ESR_mon_R4 monitores up to 4 Real inputs and reports changes with time stamd and adress label.
the module checks 4 inputs for a change of more than the specified sensitivity S and reports all changes with time and adress stamp to the output.

*)
(* read system timer *)
tx := DWORD_TO_TIME(T_PLC_MS());
P0 := ADR(R0);
P1 := ADR(R1);
P2 := ADR(R2);
P3 := ADR(R3);

ESR_Flag := FALSE;
esr_out[3].typ := 0;
esr_out[2].typ := 0;
esr_out[1].typ := 0;
esr_out[0].typ := 0;
cnt := 0;

(* check if inputs have chaged and fill buffer *)
IF DIFFER(R0,  X0, S0) THEN
	esr_out[cnt].typ := 20;
	esr_out[cnt].adress := a0;
	esr_out[cnt].DS := DT_in;
	esr_out[cnt].TS := TX;
	esr_out[cnt].data[0] := Byte_of_Dword(P0^,0);
	esr_out[cnt].data[1] := Byte_of_Dword(P0^,1);
	esr_out[cnt].data[2] := Byte_of_Dword(P0^,2);
	esr_out[cnt].data[3] := Byte_of_Dword(P0^,3);
	X0 := R0;
	cnt := cnt + 1;
	esr_flag := TRUE;
END_IF;
IF differ(R1,  X1, S1) THEN
	esr_out[cnt].typ := 20;
	esr_out[cnt].adress := a1;
	esr_out[cnt].DS := DT_in;
	esr_out[cnt].TS := TX;
	esr_out[cnt].data[0] := Byte_of_Dword(P1^,0);
	esr_out[cnt].data[1] := Byte_of_Dword(P1^,1);
	esr_out[cnt].data[2] := Byte_of_Dword(P1^,2);
	esr_out[cnt].data[3] := Byte_of_Dword(P1^,3);
	X1 := R1;
	cnt := cnt + 1;
	esr_flag := TRUE;
END_IF;
IF differ(R2,  X2, S2) THEN
	esr_out[cnt].typ := 20;
	esr_out[cnt].adress := a2;
	esr_out[cnt].DS := DT_in;
	esr_out[cnt].TS := TX;
	esr_out[cnt].data[0] := Byte_of_Dword(P2^,0);
	esr_out[cnt].data[1] := Byte_of_Dword(P2^,1);
	esr_out[cnt].data[2] := Byte_of_Dword(P2^,2);
	esr_out[cnt].data[3] := Byte_of_Dword(P2^,3);
	X2 := R2;
	cnt := cnt + 1;
	esr_flag := TRUE;
END_IF;
IF DIFFER(R3,  X3, S3) THEN
	esr_out[cnt].typ := 20;
	esr_out[cnt].adress := a3;
	esr_out[cnt].DS := DT_in;
	esr_out[cnt].TS := TX;
	esr_out[cnt].data[0] := Byte_of_Dword(P3^,0);
	esr_out[cnt].data[1] := Byte_of_Dword(P3^,1);
	esr_out[cnt].data[2] := Byte_of_Dword(P3^,2);
	esr_out[cnt].data[3] := Byte_of_Dword(P3^,3);
	X3 := R3;
	cnt := cnt + 1;
	esr_flag := TRUE;
END_IF;


(* revision history
hm	26. jan 2007	rev 1.0
	original version

hm	17. sep. 2007		rev 1.1
	replaced time() with T_PLC_MS() for compatibility reasons

hm	8. dec. 2007		rev 1.2
	corrected an error while esr typ would not be set

hm	16. mar. 2008		rev 1.3
	deleted wrong conversion real_to_dword

*)
END_FUNCTION_BLOCK

(* POU ESR_MON_X8, ST *)
FUNCTION_BLOCK ESR_MON_X8
VAR_INPUT
	s0, s1, s2, s3, s4, s5, s6, s7 : BYTE;
	DT_in : DT;
	Mode : BYTE := 3;
END_VAR
VAR_INPUT CONSTANT
	a0, a1, a2, a3, a4, a5, a6, a7 : STRING(10);
END_VAR
VAR_OUTPUT
	ESR_Out: ARRAY [0..3] OF esr_data;
	ESR_Flag : BOOL;
END_VAR
VAR
	x0, x1, x2, x3, x4, x5, x6, x7 : BYTE;
	tx: TIME;
	cnt : INT;
END_VAR

(*
version 1.1	17 sep 2007
programmer 	hugo
tested by		tobias

ESR_MON_X8 is a status and error collector.
the module checks 8 status inputs for a change and reports up to 4 input changes with time and adress stamp to the output.
the mode can be 
1 for error only
2 for error and status
3 for error, status and debug
the adress label of the 8 inputs can be configured individually.
*)
(* read system timer *)
tx := DWORD_TO_TIME(T_PLC_MS());

ESR_Flag := FALSE;
esr_out[3].typ := 0;
esr_out[2].typ := 0;
esr_out[1].typ := 0;
esr_out[0].typ := 0;
cnt := 0;


(* check if inputs have chaged and fill buffer *)
IF s0 <> X0 AND ((s0 < 100) OR (S0 > 99 AND S0 < 200 AND mode >= 2) OR (S0 > 199 AND mode = 3)) THEN
	esr_out[cnt] := status_to_ESR(s0, a0, DT_in, TX);
	X0 := S0;
	cnt := cnt + 1;
	esr_flag := TRUE;
END_IF;
IF s1 <> X1 AND ((s1 < 100) OR (S1 > 99 AND S1 < 200 AND mode >= 2) OR (S1 > 199 AND mode = 3)) THEN
	esr_out[cnt] := status_to_ESR(s1, a1, DT_in, TX);
	X1 := S1;
	cnt := cnt + 1;
	esr_flag := TRUE;
END_IF;
IF s2 <> X2 AND ((s2 < 100) OR (S2 > 99 AND S2 < 200 AND mode >= 2) OR (S2 > 199 AND mode = 3)) THEN
	esr_out[cnt] := status_to_ESR(s2, a2, DT_in, TX);
	X2 := S2;
	cnt := cnt + 1;
	esr_flag := TRUE;
END_IF;
IF s3 <> X3 AND ((s3 < 100) OR (S3 > 99 AND S3 < 200 AND mode >= 2) OR (S3 > 199 AND mode = 3)) THEN
	esr_out[cnt] := status_to_ESR(s3, a3, DT_in, TX);
	X3 := S3;
	cnt := cnt + 1;
	esr_flag := TRUE;
END_IF;
IF cnt < 4 AND s4 <> X4 AND ((s4 < 100) OR (S4 > 99 AND S4 < 200 AND mode >= 2) OR (S4 > 199 AND mode = 3)) THEN
	esr_out[cnt] := status_to_ESR(s4, a4, DT_in, TX);
	X4 := S4;
	cnt := cnt + 1;
	esr_flag := TRUE;
END_IF;
IF cnt < 4 AND s5 <> X5 AND ((s5 < 100) OR (S5 > 99 AND S5 < 200 AND mode >= 2) OR (S5 > 199 AND mode = 3)) THEN
	esr_out[cnt] := status_to_ESR(s5, a5, DT_in, TX);
	X5 := S5;
	cnt := cnt + 1;
	esr_flag := TRUE;
END_IF;
IF cnt < 4 AND s6 <> X6 AND ((s6 < 100) OR (S6 > 99 AND S6 < 200 AND mode >= 2) OR (S6 > 199 AND mode = 3)) THEN
	esr_out[cnt] := status_to_ESR(s6, a6, DT_in, TX);
	X6 := S6;
	cnt := cnt + 1;
	esr_flag := TRUE;
END_IF;
IF cnt < 4 AND s7 <> X7 AND ((s7 < 100) OR (S7 > 99 AND S7 < 200 AND mode >= 2) OR (S7 > 199 AND mode = 3)) THEN
	esr_out[cnt] := status_to_ESR(s7, a7, DT_in, TX);
	X7 := S7;
	cnt := cnt + 1;
	esr_flag := TRUE;
END_IF;


(* revision history
hm	26. jan 2007		rev 1.0
	original version

hm	17. sep 2007	rev 1.1
	replaced time() with T_PLC_MS() for compatibility reasons
	
*)
END_FUNCTION_BLOCK

(* POU STATUS_TO_ESR, ST *)
FUNCTION STATUS_TO_ESR : esr_data
VAR_INPUT
	status : BYTE;
	adress : STRING(10);
	DT_in : DT;
	TS : TIME;
END_VAR
VAR
END_VAR

(*
version 1.0	6 oct 2006
programmer 	hugo
tested by		tobias

status_to_esr creates esr data from a status byte.

*)
IF status < 100 THEN
	status_to_ESR.typ := 1;
ELSIF status < 200 THEN
	status_to_ESR.typ := 2;
ELSE
	status_to_ESR.typ := 3;
END_IF;
status_to_ESR.adress:= adress;
status_to_ESR.DS := DT_in;
status_to_ESR.TS := TS;
status_to_ESR.data[0] := status;
END_FUNCTION

(* POU EXEC, ST *)
FUNCTION EXEC : STRING(STRING_LENGTH)
VAR_INPUT
	str : STRING(STRING_LENGTH);
END_VAR
VAR
	pos: INT;
	R1: REAL;
	R2: REAL;
	operator: STRING(10);
END_VAR

(*
version 1.4	29. mar. 2008
programmer 	hugo
tested by		tobias

exec executes a mathematical term and returns the result as a string
the term can only be a simple term without brackets and only one operator
allowed operastors are: (+, -, *, /, ^, sqrt, sin, cos, tan).

*)
(* extract both numbers and operator *)
EXEC := UPPERCASE(TRIM(str));

pos := FINDB_NONUM(EXEC);
IF pos > 1 THEN R1 := STRING_TO_REAL(LEFT(EXEC,pos-1)); END_IF;
R2 := STRING_TO_REAL(RIGHT(EXEC,LEN(EXEC)-pos));
EXEC := LEFT(EXEC,pos);
pos := FINDB_NUM(EXEC);
operator := RIGHT(EXEC,LEN(EXEC) - pos);
IF operator = '' AND LEN(str) = 0 THEN
	EXEC := '';
	RETURN;
ELSIF operator = '' THEN
	EXEC := str;
	RETURN;
END_IF;
IF operator = '^' THEN
	EXEC := REAL_TO_STRING(EXPT(R1, R2));
ELSIF operator = 'SQRT' THEN
	EXEC := REAL_TO_STRING(SQRT(R2));
ELSIF operator = 'SIN' THEN
	EXEC := REAL_TO_STRING(SIN(r2));
ELSIF operator = 'COS' THEN
	EXEC := REAL_TO_STRING(COS(r2));
ELSIF operator = 'TAN' THEN
	EXEC := REAL_TO_STRING(TAN(R2));
ELSIF operator = '*' THEN
	EXEC := REAL_TO_STRING(R1 * R2);
ELSIF operator = '/' THEN
	IF R2 <> 0 THEN EXEC := REAL_TO_STRING(R1 / R2); ELSE EXEC := 'ERROR'; END_IF;
ELSIF operator = '+' THEN
	EXEC := REAL_TO_STRING(r1 + r2);
ELSIF operator = '-' THEN
	EXEC := REAL_TO_STRING(r1 - r2);
ELSE
	EXEC := 'ERROR';
END_IF;

IF EXEC = 'ERROR' THEN
	RETURN;
(* some systems deliver integer instead of real *)
ELSIF FIND(EXEC,'.') = 0 THEN
	EXEC := CONCAT(EXEC, '.0');
(* some systems deliver n. instead of n.0 ! *)
ELSIF RIGHT(EXEC,1) = '.' THEN
	EXEC := CONCAT(EXEC,'0');
END_IF;


(* revision history

hm 	6.feb 2007		rev 1.1
	cos has to be written in uppercase
	divide by 0 will return an error

hm	5. mar. 2008	rev 1.2
	add a 0 to the string if a '.' is at the end of the string

hm	20. mar. 2008	rev 1.3
	make sure the function always returns a real value in the form of x.y

hm	29. mar. 2008	rev 1.4
	changed STRING to STRING(STRING_LENGTH)
*)
END_FUNCTION

(* POU UPPERCASE, ST *)
FUNCTION UPPERCASE : STRING(STRING_LENGTH)
VAR_INPUT
	str : STRING(STRING_LENGTH);
END_VAR
VAR
	pt : POINTER TO BYTE;
	pos: INT;
	l: INT;
END_VAR

(*
version 1.3	29. mar. 2008
programmer 	hugo
tested by	tobias

uppercase returns str while all letters a..z and ä,ö,ü are converted to uppercase

*)
pt := ADR(UPPERCASE);
UPPERCASE := str;
l := LEN(str);
FOR pos := 1 TO l DO
	pt^ := TO_UPPER(pt^);
	pt := pt + 1;
END_FOR;

(* revision histroy
hm	6. oct. 2006	rev 1.0
	original release

hm	4. feb. 2008	rev 1.1
	improved performance
	added Ä,Ö,Ü

hm	6. mar. 2008	rev 1.2
	added support for exteded Ascii

hm	29. mar. 2008	rev 1.3
	changed STRING to STRING(STRING_LENGTH)

*)	
END_FUNCTION

(* POU TRIM, ST *)
FUNCTION TRIM : STRING(STRING_LENGTH)
VAR_INPUT
	str : STRING(STRING_LENGTH);
END_VAR
VAR
	pos: INT;
END_VAR

(*
version 1.2	29. mar. 2008
programmer 	hugo
tested by	tobias

the function deletes all blanks within a string.

*)
TRIM := str;
REPEAT
	pos := FIND(trim,' ');
	IF pos > 0 THEN TRIM := REPLACE(TRIM,'',1,pos); END_IF;
UNTIL pos = 0	END_REPEAT;


(* revision histroy
hm	6.10.2006		rev 1.0
	original release

hm	20. mar. 2008	rev 1.1
	avoid to call replace with pos = 0 because some systems will produce an error

hm	29. mar. 2008	rev 1.2
	changed STRING to STRING(STRING_LENGTH)
*)
END_FUNCTION

(* POU FINDB_NONUM, ST *)
FUNCTION FINDB_NONUM : INT
VAR_INPUT
	str : STRING(STRING_LENGTH);
END_VAR
VAR
	pos: INT;
	pt : POINTER TO BYTE;
END_VAR

(*
version 1.3	21. oct. 2008
programmer 	hugo
tested by	oscat

findB_noNum searches str backwards and returns the last position which is not a number.
a number is characterized by a letter "0..9" or "."

*)
pt := ADR(str) + LEN(str) - 1;
FOR pos := LEN(str) TO 1 BY -1 DO;
	IF (PT^ < 48 AND PT^ <> 46) OR PT^ > 57 THEN
		FINDB_NONUM := pos;
		RETURN;
	END_IF;
	PT := PT - 1;
END_FOR;
FINDB_NONUM := 0;


(* revision history
hm	6. oct 2006		rev 1.0
	original version

hm	29. feb 2008	rev 1.1
	improved performance

hm	29. mar. 2008	rev 1.2
	changed STRING to STRING(STRING_LENGTH)

hm	21. oct. 2008	rev 1.3
	optimized code
*)
END_FUNCTION

(* POU FINDB_NUM, ST *)
FUNCTION FINDB_NUM : INT
VAR_INPUT
	str : STRING(STRING_LENGTH);
END_VAR
VAR
	pos: INT;
	pt : POINTER TO BYTE;
END_VAR

(*
version 1.2	29. mar. 2008
programmer 	hugo
tested by	tobias

findB_Num searches str backward and returns the last position of a number
a number is characterized by a letter "0..9" or "."

*)
pt := ADR(str) + LEN(str) - 1;
FOR pos := LEN(str) TO 1 BY -1 DO;
	IF (PT^ > 47 AND PT^ < 58) OR PT^ = 46 THEN
		FINDB_NUM := pos;
		RETURN;
	END_IF;
	PT := PT - 1;
END_FOR;
FINDB_NUM := 0;

(* revision history
hm	6. oct 2006		rev 1.0
	original version

hm	29. feb 2008	rev 1.1
	improved performance

hm	29. mar. 2008	rev 1.2
	changed STRING to STRING(STRING_LENGTH)
*)
END_FUNCTION

(* POU EXPN, ST *)
FUNCTION EXPN : REAL
VAR_INPUT
	X : REAL;
	N : INT;
END_VAR
VAR
	sign: BOOL;
END_VAR

(*
version 1.1	 22. oct. 2008
programmer 	hugo
tested by	oscat

this function calculates X to the power of N (Y = X^N) whilke N is an integer
especially on CPU's without a floating point unit this algorythm is about 30 times faster then the IEC standard EXPT() Function

*)
sign := n.15;
N := ABS(N);
IF N.0 THEN EXPN := X; ELSE EXPN := 1; END_IF;
N := SHR(N,1);
WHILE N > 0 DO
   X := X * X;
   IF N.0 THEN EXPN := EXPN * X; END_IF;
   N := SHR(N,1);
END_WHILE;
IF sign THEN EXPN := 1 / EXPN; END_IF;

(* old code before 1.1
IF n.15 THEN
	(* N is negative *)
	N := ABS(N);
	IF N.0 THEN expn := X; ELSE expn := 1; END_IF;
	N := SHR(N,1);
	WHILE N > 0 DO
		X := X * X;
		IF N.0 THEN expn := expn * X; END_IF;
		N := SHR(N,1);
	END_WHILE;
	expn := 1 / expn;
ELSE;
	IF N.0 THEN EXPN := X; ELSE EXPN := 1; END_IF;
	N := SHR(N,1);
	WHILE N > 0 DO
		X := X * X;
		IF N.0 THEN expn := expn * X; END_IF;
		N := SHR(N,1);
	END_WHILE;
END_IF;
*)


(* revision history
hm	4. dec 2007		rev 1.0
	original version

hm	22. oct. 2008	rev 1.1
	optimized code
*)
END_FUNCTION

(* POU F_LAMP, ST *)
FUNCTION_BLOCK F_LAMP
VAR_INPUT
	SWITCH : BOOL;
	DIMM : BYTE := 255;
	RST : BOOL;
END_VAR
VAR_OUTPUT
	LAMP : BYTE;
	STATUS : BYTE;
END_VAR
VAR_IN_OUT
	ONTIME : UDINT;
	CYCLES : UDINT;
END_VAR
VAR_INPUT CONSTANT
	T_NO_DIMM : UINT := 100;
	T_MAINTENANCE : UINT := 15000;
END_VAR
VAR
	runtime : ONTIME;
END_VAR

(*
version 1.2	22. oct. 2008
programmer 	hugo
tested by	oscat

F_Lamp is an interface to flourescent lamps. its main purpose is to protect flourescent lamps from dimming within the first T_NO_DIMM Time.
If Flourescent Lamps are dimmed during the first 100 hours the lifetime of the lamp is reduced dramatically.
The interface also counts ontime and cycles of the lamp for maintanance purposes.

*)
runtime(in := switch, seconds := ontime, cycles := cycles);

IF RST THEN
	ONTIME := 0;
	CYCLES := 0;
END_IF;
IF SWITCH THEN
	IF ontime < T_NO_DIMM * 3600 THEN
		LAMP := 255;
		STATUS := 111;
	ELSE
		LAMP := DIMM;
		STATUS := 112;
	END_IF;
ELSE
	LAMP := 0;
	STATUS := 110;
END_IF;


IF ontime >= T_maintenance * 3600 AND T_Maintenance > 0 THEN
	status := 120;
END_IF;



(* revision history
hm	8. feb. 2007	rev 1.1
	original version

hm	22. oct. 2008	rev 1.2
	changed use of ontime for ontime 2.0
	ontime is now in seconds not hours
*)
END_FUNCTION_BLOCK

(* POU F_LIN, ST *)
FUNCTION F_LIN : REAL
VAR_INPUT
	X : REAL;
	A : REAL;
	B : REAL;
END_VAR
VAR
END_VAR

(*
version 1.0	1 sep 2006
programmer 	hugo
tested by		tobias

this function calculates the linear equation f_lin = a*x + b

*)
F_lin := A * X + B;
END_FUNCTION

(* POU F_LIN2, ST *)
FUNCTION F_LIN2 : REAL
VAR_INPUT
	X : REAL;
	X1: REAL;
	Y1 : REAL;
	X2 : REAL;
	Y2 : REAL;
END_VAR
VAR

END_VAR

(*
version 1.0	1 jan 2007
programmer 	hugo
tested by		tobias

this function calculates the linear equation f_lin = a*x + b given by two points x1/y1 and x2/y2.

*)
F_LIN2 := (Y2 - Y1) / (X2 - X1) * (X - X1) + Y1;


(* revision history
hm	1. jan. 2007	rev 1.0
	original release

hm	17. dec. 2008	rev 1.1
	optimized formula

*)
END_FUNCTION

(* POU F_POLY, ST *)
FUNCTION F_POLY : REAL
VAR_INPUT
	X : REAL;
	C : ARRAY[0..7] OF REAL;
END_VAR
VAR
	x2: REAL;
	X4 : REAL;
	X6: REAL;
END_VAR

(*
version 1.0	20. may. 2008
programmer 	hugo
tested by		tobias

this function calculates the polynom C[0] + C[1]*X^1 + C[2]*X^2 * C[3]*X^3 + C[4]*X^4 + C[5]*X^5 + C[6]*X^6 + C[7]*X^7

*)
x2 := X * X;
X4 := X2 * X2;
X6 := X4 * X2;
F_POLY := C[7] * X6 * X + C[6] * X6 + C[5] * X4 * X + C[4] * X4 + c[3] * X2*X + C[2] * X2 + C[1] * X + C[0];


(* revision history
hm		20. may. 2008		rev 1.0
	original version

*)
END_FUNCTION

(* POU F_POWER, ST *)
FUNCTION F_POWER : REAL
VAR_INPUT
	a : REAL;
	x : REAL;
	n : REAL;
END_VAR
VAR
END_VAR

(*
version 1.0	1 sep 2006
programmer 	hugo
tested by		tobias

this function calculates the power equation f_power = a*x^n

*)
F_power := a * EXPT(X,N);
END_FUNCTION

(* POU F_QUAD, ST *)
FUNCTION F_QUAD : REAL
VAR_INPUT
	X : REAL;
	A : REAL;
	B : REAL;
	C : REAL;
END_VAR
VAR
END_VAR

(*
version 1.0	1 sep 2006
programmer 	hugo
tested by		tobias

this function calculates the quadratic equation f_lin = a*x + b

*)
F_quad := a * X * X + B * X + C;
END_FUNCTION

(* POU F_TO_C, ST *)
FUNCTION F_TO_C : REAL
VAR_INPUT
	fahrenheit : REAL;
END_VAR
VAR
END_VAR

(*
version 1.1	6. jan 2008
programmer 	hugo
tested BY		tobias

this FUNCTION converts fahrenheit TO celsius

executioin TIME on wago 750-841 = 15us
*)
F_to_C := (fahrenheit -32) * 0.5555555555555;

(* revision history
hm	4. aug 2006		rev 1.0
	original version

hm	6. jan 2008		rev 1.1
	improved performance

*)
END_FUNCTION

(* POU F_TO_OM, ST *)
FUNCTION F_TO_OM : REAL
VAR_INPUT
	F : REAL;
END_VAR
VAR
END_VAR

(*
version 1.1	18. oct. 2008
programmer 	hugo
tested by	oscat

this function converts frequency to Omega F
Omega = 2*PI*F
*)
F_TO_OM := math.PI2 * F;


(* revision history
hm	22. jan. 2007	rev 1.0
	original version

hm	18. oct. 2008	rev 1.1
	unsing math constants

*)
END_FUNCTION

(* POU F_TO_PT, ST *)
FUNCTION F_TO_PT : TIME
VAR_INPUT
	F : REAL;
END_VAR
VAR
END_VAR

(*
version 1.0	4 aug 2006
programmer 	hugo
tested by		tobias

this function converts frequency to periode time  
*)
F_to_PT := DWORD_TO_TIME(REAL_TO_DWORD(1/F*1000));
END_FUNCTION

(* POU FACT, ST *)
FUNCTION FACT : DINT
VAR_INPUT
	X : INT;
END_VAR
VAR
	i: INT;
END_VAR

(*
version 1.4	27. 0ct. 2008
programmer 	hugo
tested by		tobias

this function calculates the factorial of x

if the input is negative or higher then 7 the output will be -1.

*)
IF X <= 5 THEN
	FACT := 1;
	FOR i := 2 TO x DO
		FACT := FACT * i;
	END_FOR;
ELSIF x <= 9 THEN
	FACT := 720;
	FOR i := 7 TO x DO
		FACT := FACT * i;
	END_FOR;
ELSIF x <= 13 THEN
	FACT := 3628800;
	FOR i := 11 TO x DO
		FACT := FACT * i;
	END_FOR;
ELSE
	FACT := -1;
END_IF;



(* code for rev 1.3
IF x >= 0 AND x < 13 THEN
	FACT := 1;
	i := 2;
	WHILE i <= x DO
		FACT := FACT * i;
		i := i + 1;
	END_WHILE;
ELSE
	FACT := -1;
END_IF;
*)


(* revision history
hm 	4.3.2007		rev 1.1
	changed a critical error where while loop was indefinite.

hm	10.12.2007		rev 1.2
	start value for i has changed to 2 for better performance

hm	10. mar 2008	rev 1.3
	changed output of fact to dint to allow bigger values

hm	27. oct. 2008	rev 1.4
	optimized code
*)
END_FUNCTION

(* POU FADE, ST *)
FUNCTION_BLOCK FADE
VAR_INPUT
	IN1 : REAL;
	IN2 : REAL;
	F : BOOL;
	TF : TIME;
	rst : BOOL;
END_VAR
VAR_OUTPUT
	Y : REAL;
END_VAR
VAR CONSTANT
	FF : WORD := 65535;
END_VAR
VAR
	rmx : RMP_W;
END_VAR

(*
version 1.2	17. de3c. 2008
programmer 	oscat
tested BY	oscat

FADE is used to crossfade between the inputs IN1 and IN2. The fade_over time is specified with TF.
When F = TRUE then Y = IN2 after the time TF, and when F = FALSE then Y = IN1.

*)
rmx(rst := rst AND NOT F, set := rst AND F, pt := TF, up := F);
Y := (in2 - In1) / 65535.0 * WORD_TO_REAL(rmx.out) + in1;


(* code for rev 1.1
IF rst THEN
	rmx(set := F, rst := NOT F);
ELSIF F AND (NOT rmx.high) THEN
	rmx(PT := TF, UP := TRUE, e := TRUE, rst := FALSE, set := FALSE);
ELSIF (NOT F) AND (NOT rmx.low) THEN
	rmx(PT := TF, UP := FALSE, e := TRUE, rst := FALSE, set := FALSE);
ELSE
	rmx(e := FALSE, rst := FALSE, set := FALSE);
END_IF;
Y := (WORD_TO_REAL(rmx.out) * in1 + WORD_TO_REAL(FF - rmx.out) * IN2) / FF;
*)


(* revision history
hm	26. dec 2007	rev 1.0
	original version

hm	18. oct. 2008	rev 1.1
	improved performance
	changed calls for rmp_w because rmp_w has chaged

hm	17. dec. 2008	rev 1.2
	function of input f was inverted

*)
END_FUNCTION_BLOCK

(* POU RMP_W, ST *)
FUNCTION_BLOCK RMP_W
VAR_INPUT
	SET : BOOL;
	PT : TIME;
	E : BOOL := TRUE;
	UP : BOOL := TRUE;
	RST : BOOL;
END_VAR
VAR_OUTPUT
	out : WORD;
	busy : BOOL;
	high : BOOL;
	low : BOOL;
END_VAR
VAR
	rmp : _RMP_W;
END_VAR

(*
version 2.0	23. oct. 2008
programmer 	oscat
tested BY	oscat

this ramp generator generates a Word wide ramp with 65535 steps
the generator has an asynchronous set and reset
the ramp is controlled by PT which is the total ramp time for a full sweep from 0..65535
an UD input controlls the direction Up or Down and the E input enables the ramp generation
a busy output indicates that the ramp is running, busy false means output is stable.
the outputs low and high will be true when the output has reached its max or min value.
*)
(* generate ramp *)
rmp(dir := UP, E := E, TR := PT, rmp := out);

(* set or reset operation *)
IF RST THEN
	out := 0;
ELSIF SET THEN
	out := 65535;
END_IF;

(* checks for outputs stable and reset or set busy flag *)
low := out = 0;
high := out = 65535;
busy := NOT (low OR high) AND E;


(* revision history:

hm 4.10.2006		rev 1.1
	added the busy output which signals that the ramp is running.

hm 22.1.2007		rev 1.2
	deleted unused variable step

hm	17.9.2007		rev 1.3
	replaced time() with t_plc_ms() for compatibility reasons

hm	28. sep 2007	rev 1.4
	added outputs on and off
	busy is now disabled while en is false
	new coding for higher accuracy and performance

hm	5. oct 2007	rev 1.5
	added statements to allow for PT to be t#0s output jumps to max or min immediately

hm	2. dec 2007	rev 1.6
	corrected an error in calculation of step response

hm	25. dec 2007	rev 1.7
	corrected an error while step response was too slow for fast rise times

hm	16. oct. 2008	rev 1.8
	improved performance

hm	18. oct. 2008	rev 1.9
	renamed inout EN to E for compatibility reasons

hm	23. oct. 2008	rev 2.0
	new code using _RMP_W
*)
END_FUNCTION_BLOCK

(* POU FF_D2E, ST *)
FUNCTION_BLOCK FF_D2E
VAR_INPUT
	D0 : BOOL;
	D1 : BOOL;
	CLK : BOOL;
	RST : BOOL;
END_VAR
VAR_OUTPUT
	Q0 : BOOL;
	Q1 : BOOL;
END_VAR
VAR
	edge : BOOL;
END_VAR

(*
version 1.2	30. oct. 2008
programmer 	hugo
tested by	oscat

dual D-type flip flop with reset and rising clock trigger

*)
IF rst THEN
	Q0 := Q1 := FALSE;
ELSIF clk AND NOT edge THEN
	Q0 := D0;
	Q1 := D1;
END_IF;
edge := CLK;

(* revision history
hm	25. dec 2007	rev 1.0
	original version

hm	27. dec 2007	rev 1.1
	changed code for better performance

hm	30. oct. 200	rev 1.2
	deleted unnecessary init with 0
*)
END_FUNCTION_BLOCK

(* POU FF_D4E, ST *)
FUNCTION_BLOCK FF_D4E
VAR_INPUT
	D0 : BOOL;
	D1 : BOOL;
	D2 : BOOL;
	D3 : BOOL;
	CLK : BOOL;
	RST : BOOL;
END_VAR
VAR_OUTPUT
	Q0 : BOOL;
	Q1 : BOOL;
	Q2 : BOOL;
	Q3 : BOOL;
END_VAR
VAR
	edge : BOOL;
END_VAR


(*
version 1.2	30. oct. 2008
programmer 	hugo
tested by	oscat

quad D-type flip flop with reset and rising clock trigger

*)
IF rst THEN
	Q0 := Q1 := Q2 := Q3 := FALSE;
ELSIF clk AND NOT edge THEN
	Q0 := D0;
	Q1 := D1;
	Q2 := D2;
	Q3 := D3;
END_IF;
edge := CLK;

(* revision history
hm	4. aug 2006		rev 1.0
	original version

hm	27. dec 2007	rev 1.1
	changed code for better performance

hm	30. oct. 200	rev 1.2
	deleted unnecessary init with 0

*)
END_FUNCTION_BLOCK

(* POU FF_DRE, ST *)
FUNCTION_BLOCK FF_DRE
VAR_INPUT
	SET : BOOL;
	D : BOOL;
	CLK : BOOL;
	RST : BOOL;
END_VAR
VAR_OUTPUT
	Q : BOOL;
END_VAR
VAR
	edge : BOOL;
END_VAR


(*
version 1.2	30. oct. 2008
programmer 	hugo
tested by	oscat

D-type flip flop with set, reset and rising clock trigger

*)
IF rst OR set THEN
	Q := NOT rst;
ELSIF clk AND NOT edge THEN
	Q := D;
END_IF;
edge := CLK;

(* revision history
hm	4. aug 2006		rev 1.0
	original version

hm	27. dec 2007	rev 1.1
	changed code for better performance

hm	30. oct. 2008	rev 1.2
	optimized performance
*)
END_FUNCTION_BLOCK

(* POU FF_JKE, ST *)
FUNCTION_BLOCK FF_JKE
VAR_INPUT
	SET : BOOL;
	J : BOOL;
	CLK : BOOL;
	K : BOOL;
	RST : BOOL;
END_VAR
VAR_OUTPUT
	Q : BOOL;
END_VAR
VAR
	edge : BOOL;
END_VAR


(*
version 1.2	30. oct. 2008
programmer 	hugo
tested by	oscat

JK-type flip flop with set, reset and rising clock trigger
set and reset are asynchron while the FF is rising edge triggered
J=0 and K=0 and CLK >>> no action
J=1 and K=0 and CLK >>> output = 1
J=0 and K=1 and CLK >>> output = 0
J=1 and K=1 and CLK >>> toggle output


*)
IF rst OR set THEN
	Q := NOT rst;
ELSIF clk AND NOT edge THEN
	IF J XOR K THEN Q := J;
	ELSE Q := K XOR Q;
	END_IF;
END_IF;
edge := CLK;

(* revision history
hm	4. aug 2006		rev 1.0
	original version

hm	27. dec 2007	rev 1.1
	changed code for better performance

hm	30. oct. 2008	rev 1.2
	optimized performance
*)
END_FUNCTION_BLOCK

(* POU FIB, ST *)
FUNCTION FIB : DINT
VAR_INPUT
	X : INT;
END_VAR
VAR
	t1, t2: DINT;
END_VAR

(*
version 1.3	26. mar. 2008
programmer 	hugo
tested by		tobias

this function calculates the fibonacci sequence

*)
IF X < 0 OR X > 46 THEN
	FIB := -1;
ELSIF x < 2 THEN
	FIB := X;
	RETURN;
ELSE
	(* the fibonacci number is the sum of the two suceeding fibonaci numbers *)
	(* we store the numbers alternatively in t1 and t2 depending on pt *)
	t2 := 1;
	WHILE X > 3 DO
		X := X-2;
		t1 := t1 + t2;
		t2 := t1 + t2;
	END_WHILE;
	IF X > 2 THEN t1 := t1 + t2; END_IF;
	fib := t1 + t2;
END_IF;

(* alternative code for very big numbers

IF X < 31 THEN
	fib := 0.4472136 * (expn(1.618034,X) - expn(-0.618034,X));
ELSE
	fib := 0.4472133 * expn(1.618034,X);
END_IF;

*)

(* revision history
hm		27. dec 2007	rev 1.0
	original version

hm		2. jan 2008	rev 1.1
	deleted unused variable pt

hm		10. mar 2008	rev 1.2
	changed output to dint instead of real

hm		26. mar. 2008	rev 1.3
	function now returns -1 for input < 0 or > 46

*)
END_FUNCTION

(* POU FIFO_16, ST *)
FUNCTION_BLOCK FIFO_16
VAR_INPUT
	Din : DWORD;
	WR : BOOL;
	E : BOOL;
	RST : BOOL;
END_VAR
VAR_OUTPUT
	Dout : DWORD;
	empty : BOOL := TRUE;
	full : BOOL;
END_VAR
VAR
	fifo : ARRAY[0..15] OF DWORD;
	NW : INT;
	NR : INT;
END_VAR

(*
version 1.3	27. oct. 2008
programmer 	hugo
tested by		oscat

16 Dword FIFO memory
*)
IF rst THEN
	(* asynchronous reset for the fifo *)
	NW := NR := 0;
	Dout := 0;
	empty := TRUE;
	full := FALSE;
ELSIF E THEN
	IF WR AND NOT full THEN
		(* write action *)
		fifo[NW] := Din;
		NW := INC1(NW, 16);
		full := NW = NR;
		empty := FALSE;
	ELSIF NOT WR AND NOT empty THEN
		(* read from stack *)
		Dout := fifo[NR];
		NR := INC1(NR, 16);
		empty := NR = NW;
		full := FALSE;
	END_IF
END_IF;

(* revision history
hm	4. aug. 2006	rev 1.0
	original version

hm	19. feb 2008	rev 1.1
	performance improvements

hm	17. oct. 2008	rev 1.2
	improved performance

ks	27. oct. 2008	rev 1.3
	optimized coding
*)
END_FUNCTION_BLOCK

(* POU FIFO_32, ST *)
FUNCTION_BLOCK FIFO_32
VAR_INPUT
	Din : DWORD;
	WR : BOOL;
	E : BOOL;
	RST : BOOL;
END_VAR
VAR_OUTPUT
	Dout : DWORD;
	empty : BOOL := TRUE;
	full : BOOL;
END_VAR
VAR
	fifo : ARRAY[0..31] OF DWORD;
	NW : INT;
	NR : INT;
END_VAR

(*
version 1.3	27. oct. 2008
programmer 	hugo
tested by		oscat

32 Dword FIFO memory
*)
IF rst THEN
	(* asynchronous reset for the fifo *)
	NW := NR := 0;
	Dout := 0;
	empty := TRUE;
	full := FALSE;
ELSIF E THEN
	IF WR AND NOT full THEN
		(* write action *)
		fifo[NW] := Din;
		NW := INC1(NW, 32);
		full := NW = NR;
		empty := FALSE;
	ELSIF NOT WR AND NOT empty THEN
		(* read from stack *)
		Dout := fifo[NR];
		NR := INC1(NR, 32);
		empty := NR = NW;
		full := FALSE;
	END_IF;
END_IF;

(* revision history
hm	4. aug. 2006	rev 1.0
	original version

hm	19. feb 2008	rev 1.1
	performance improvements

hm	17. oct. 2008	rev 1.2
	improved performance

ks	27. oct. 2008 rev 1.3
	improved code
*)
END_FUNCTION_BLOCK

(* POU FILTER_DW, ST *)
FUNCTION_BLOCK FILTER_DW
VAR_INPUT
	X : DWORD;
	T : TIME;
END_VAR
VAR_OUTPUT
	Y : DWORD;
END_VAR
VAR
	last : DWORD;
	tx: DWORD;
	init: BOOL;
	Yi : REAL;
END_VAR

(*
version 1.1	3. nov. 2008
programmer 	hugo
tested by	oscat

FILTER_DW is an low pass filter with a programmable time T used for DWORD format.
 
*)
(* read system time *)
tx := T_PLC_MS();

(* startup initialisation *)
IF NOT init OR T = t#0s THEN
	init := TRUE;
	Yi := DWORD_TO_REAL(X);
ELSE
	Yi := Yi + (DWORD_TO_REAL(X) - DWORD_TO_REAL(Y)) * DWORD_TO_REAL(tx - last) / TIME_TO_REAL(T);
END_IF;
last := tx;

Y := REAL_TO_DWORD(Yi);



(*
hm 10. oct. 2008	rev 1.0
	original version

hm	3. nov. 2008	REV 1.1
	corrected an overflow problem
*)
END_FUNCTION_BLOCK

(* POU FILTER_I, ST *)
FUNCTION_BLOCK FILTER_I
VAR_INPUT
	X : INT;
	T : TIME;
END_VAR
VAR_OUTPUT
	Y : INT;
END_VAR
VAR
	Yi : DINT;
	last : DWORD;
	tx: DWORD;
	init: BOOL;
END_VAR

(*
version 1.0	8. nov. 2008
programmer 	hugo
tested by	oscat

FILTER_I is a low pass filter with a programmable time T used for INT format.
 
*)
(* read system time *)
tx := T_PLC_MS();

(* startup initialisation *)
IF NOT init OR T = t#0s THEN
	init := TRUE;
	Yi := INT_TO_DINT(X) * 1000;
ELSE
	(* to increase accuracy of the filter we calculate internal Yi wich is Y * 1000 *)
	Yi := Yi + INT_TO_DINT(X - Y) * DWORD_TO_DINT(tx - last) * 1000 / TIME_TO_DINT(T);
END_IF;
last := tx;
Y := DINT_TO_INT(yi / 1000);



(*
hm 8. nov. 2008	rev 1.0
	original version

*)
END_FUNCTION_BLOCK

(* POU FILTER_MAV_DW, ST *)
FUNCTION_BLOCK FILTER_MAV_DW
VAR_INPUT
	X : DWORD;
	N : UINT;
	RST : BOOL;
END_VAR
VAR_OUTPUT
	Y : DWORD;
END_VAR
VAR
	init: BOOL;
	buffer : ARRAY[0..31] OF DWORD;
	i: INT;
END_VAR
VAR_TEMP
	tmp: INT;
END_VAR

(*
version 1.2	24. nov. 2008
programmer 	hugo
tested by	oscat

FILTER_MAV_DW is a moving average filter with programmable length N for DWORD Data.
 
*)
(* startup initialisation *)
IF NOT init OR rst OR N = 0 THEN
	init := TRUE;
	tmp := UINT_TO_INT(N)-1;
	FOR i := 0 TO tmp DO
		buffer[i] := X;
	END_FOR;
	Y := X;
ELSE
	i := INC1(i, UINT_TO_INT(N));
	Y := Y + (X - buffer[i]) / N;
	buffer[i] := X;
END_IF;




(*
hm 13. oct. 2008	rev 1.0
	original version

hm	27. oct. 2008	rev 1.1
	added typecast to avoid warnings

hm	24. nov. 2008	rev 1.2
	added typecasts to avoid warnings
	avoid divide by 0 if N = 0

*)
END_FUNCTION_BLOCK

(* POU FILTER_MAV_W, ST *)
FUNCTION_BLOCK FILTER_MAV_W
VAR_INPUT
	X : WORD;
	N : UINT;
	RST : BOOL;
END_VAR
VAR_OUTPUT
	Y : WORD;
END_VAR
VAR
	init: BOOL;
	buffer : ARRAY[0..31] OF WORD;
	i: INT;
END_VAR
VAR_TEMP
	tmp : INT;
END_VAR

(*
version 1.2	24. nov. 2008
programmer 	hugo
tested by	oscat

FILTER_MAV_W is a moving average filter with programmable length N for WORD Data.
 
*)
(* startup initialisation *)
IF NOT init OR rst OR N = 0 THEN
	init := TRUE;
	tmp := UINT_TO_INT(N) - 1;
	FOR i := 0 TO tmp DO
		buffer[i] := X;
	END_FOR;
	Y := X;
ELSE
	i := INC1(i, UINT_TO_INT(N));
	Y := Y + (X - buffer[i]) / N;
	buffer[i] := X;
END_IF;



(*
hm 13. oct. 2008	rev 1.0
	original version

hm	18. oct. 2008	rev 1.1
	added typecast to avoid warnings

hm	24. nov. 2008	rev 1.2
	added typecasts to avoid warnings
	avoid devide by 0 if N = 0
*)
END_FUNCTION_BLOCK

(* POU FILTER_W, ST *)
FUNCTION_BLOCK FILTER_W
VAR_INPUT
	X : WORD;
	T : TIME;
END_VAR
VAR_OUTPUT
	Y : WORD;
END_VAR
VAR
	last : DWORD;
	tx: DWORD;
	init: BOOL;
END_VAR

(*
version 1.1	3. nov. 2008
programmer 	hugo
tested by	oscat

FILTER_W is an low pass filter with a programmable time T used for WORD format.
 
*)
(* read system time *)
tx := T_PLC_MS();

(* startup initialisation *)
IF NOT init OR T = t#0s THEN
	init := TRUE;
	Y := X;
ELSE
	Y := Y + DINT_TO_WORD(WORD_TO_DINT(X - Y) * DWORD_TO_DINT(tx-last) / TIME_TO_DINT(T));
END_IF;
last := tx;



(*
hm 10. oct. 2008	rev 1.0
	original version

hm	3. nov. 2008	rev 1.1
	fixed overflow problen in formula
*)
END_FUNCTION_BLOCK

(* POU FILTER_WAV, ST *)
FUNCTION_BLOCK FILTER_WAV
VAR_INPUT
	X : REAL;
	W : ARRAY[0..15] OF REAL;
	RST : BOOL;
END_VAR
VAR_OUTPUT
	Y : REAL;
END_VAR
VAR
	init: BOOL;
	buffer : ARRAY[0..15] OF REAL;
	i: INT;
	n: INT;
END_VAR

(*
version 1.1	27. oct. 2008
programmer 	hugo
tested by	oscat

FILTER_WAV is a moving average filter with programmable length N for DWORD Data.
 
*)
(* startup initialisation *)
IF NOT init OR rst THEN
	init := TRUE;
	FOR i := 0 TO 15 DO
		buffer[i] := X;
	END_FOR;
	i := 15;
	Y := X;
ELSE
	i := INC1(i, 16);
	buffer[i] := X;
END_IF;

(* calculate the weighted average *)
Y := 0;
FOR n := 0 TO 15 DO
	Y := buffer[i] * W[n] + Y;
	i := DEC1(i, 16);
END_FOR;


(*
hm 	14. oct. 2008	rev 1.0
	original version

hm	27. oct. 2008	rev 1.1
	changed _DEC and _INC to DEC1 and INC1
*)
END_FUNCTION_BLOCK

(* POU FIND_CHAR, ST *)
FUNCTION FIND_CHAR : INT
VAR_INPUT
	str : STRING(STRING_LENGTH);
	pos : INT;
END_VAR
VAR
	i: INT;
	pt : POINTER TO ARRAY[1..255] OF BYTE;
	stop: INT;
	X: BYTE;
END_VAR

(*
version 1.3	21. oct. 2008
programmer 	hugo
tested by	tobias

find_char searches str and returns the starting position of the first character that is not a control character.
control characters are the ascii character 00 .. 31 and 127

*)
pt := ADR(str);
stop := LEN(str);
FOR i := MAX(pos,1) TO stop DO;
	X := pt^[i];
	IF X > 31 AND ((setup.EXTENDED_ASCII AND X <> 127) OR (NOT setup.EXTENDED_ASCII AND X < 127)) THEN
		FIND_CHAR := i;
		RETURN;
	END_IF;
END_FOR;
FIND_CHAR := 0;


(* revision history
hm	29. feb 2008	rev 1.0
	original version

hm	26. mar. 2008	rev 1.1
	char will now accept extended ascii

hm	29. mar. 2008	rev 1.2
	changed STRING to STRING(STRING_LENGTH)

hm	21. oct. 2008	rev 1.3
	changes setup constants
	optimized code
*)
END_FUNCTION

(* POU FIND_CTRL, ST *)
FUNCTION FIND_CTRL : INT
VAR_INPUT
	str : STRING(STRING_LENGTH);
	pos : INT;
END_VAR
VAR
	i: INT;
	pt : POINTER TO ARRAY[1..255] OF BYTE;
	stop: INT;
	x: BYTE;
END_VAR

(*
version 1.2	29. mar. 2008
programmer 	hugo
tested by		tobias

find_ctrl searches str and returns the starting position of a control character
control characters are the ascii character 00 .. 31 and 127.

*)
pt := ADR(str);
stop := LEN(str);
FOR i := MAX(pos,1) TO stop DO;
	x := PT^[I];
	IF x < 32 OR X = 127 THEN
		FIND_CTRL := i;
		RETURN;
	END_IF;
END_FOR;
FIND_CTRL := 0;


(* revision history
hm	29. feb 2008	rev 1.0
	original version

hm	26. mar. 2008	rev 1.1
	character 127 is now recognized as control

hm	29. mar. 2008	rev 1.2
	changed STRING to STRING(STRING_LENGTH)
*)
END_FUNCTION

(* POU FIND_NONUM, ST *)
FUNCTION FIND_NONUM : INT
VAR_INPUT
	str : STRING(STRING_LENGTH);
	pos : INT;
END_VAR
VAR
	i: INT;
	pt : POINTER TO ARRAY[1..255] OF BYTE;
	end: INT;
	X: BYTE;
END_VAR

(*
version 1.3	21. oct. 2008
programmer 	hugo
tested by	tobias

find_noNum searches str and returns the first position which is not a number.
a number is characterized by a letter "0..9" or "."

*)
pt := ADR(str);
end := LEN(str);
FOR i := MAX(pos,1) TO end DO;
	X := pt^[i];
	IF (X < 48 AND X <> 46) OR X > 57 THEN
		FIND_NONUM := i;
		RETURN;
	END_IF;
END_FOR;
FIND_NONUM := 0;


(* revision history
hm	6. oct. 2006	rev 1.0
	original version

hm	29. feb 2008	rev 1.1
	added input pos to start search at position

hm	29. mar. 2008	rev 1.2
	changed STRING to STRING(STRING_LENGTH)

hm	21. oct. 2008	rev 1.3
	optimized code

*)
END_FUNCTION

(* POU FIND_NUM, ST *)
FUNCTION FIND_NUM : INT
VAR_INPUT
	str : STRING(STRING_LENGTH);
	pos : INT;
END_VAR
VAR
	i : INT;
	pt : POINTER TO ARRAY[1..255] OF BYTE;
	stop : INT;
	X: BYTE;
END_VAR

(*
version 1.2	29. mar. 2008
programmer 	hugo
tested by		tobias

find_Num searches str and returns the starting position of a number
a number is characterized by a letter "0..9" or "."

*)
pt := ADR(str);
stop := LEN(str);
FOR i := MAX(pos,1) TO stop DO;
	X := pt^[i];
	IF (X > 47 AND X < 58) OR X = 46 THEN
		FIND_NUM := i;
		RETURN;
	END_IF;
END_FOR;
FIND_NUM := 0;


(* revision history
hm	6. oct. 2006	rev 1.0
	original version

hm	29. feb 2008	rev 1.1
	added input pos to start search at position

hm	29. mar. 2008	rev 1.2
	changed STRING to STRING(STRING_LENGTH)

*)
END_FUNCTION

(* POU FINDB, ST *)
FUNCTION FINDB : INT
VAR_INPUT
	str1 : STRING(STRING_LENGTH);
	str2 : STRING(STRING_LENGTH);
END_VAR
VAR
	pos: INT;
	length: INT;
END_VAR

(*
version 1.3	29. mar. 2008
programmer 	hugo
tested by		tobias

the function find searches an str1 for the presence of str2 and returns the first position of str1 of the last presence in instring.
the function is similar to find except it searches from the right to left.
 a 0 is returned if the string is not found.

*)
length := LEN(str2);
FOR pos := LEN(str1) - length + 1 TO 1 BY -1 DO
	IF MID(str1,length,pos) = str2 THEN
		FindB := pos;
		RETURN;
	END_IF;
END_FOR;
FindB := 0;

(* revision history
hm	6. oct 2006		rev 1.0
	original version

hm	15 dec 2007		rev 1.1
	changed code for better performance

hm	29. feb 2008	rev 1.2
	added findb := 0 for compatibility reasons

hm	29. mar. 2008	rev 1.3
	changed STRING to STRING(STRING_LENGTH)
*)
END_FUNCTION

(* POU LENGTH, ST *)
FUNCTION_BLOCK LENGTH
VAR_INPUT
	m : REAL;
	p : REAL;
	in : REAL;
	ft : REAL;
	yd : REAL;
	mile : REAL;
	sm : REAL;
	fm : REAL;
END_VAR
VAR_OUTPUT
	Ym : REAL;
	Yp : REAL;
	Yin : REAL;
	Yft : REAL;
	Yyd : REAL;
	Ymile : REAL;
	Ysm : REAL;
	Yfm : REAL;
END_VAR
VAR
END_VAR

(*
version 1.0	27 mar 2007
programmer 	hugo
tested by		oscat

this function converts different length units
any unused input can simply be left open.
different inputs connected at the same time will be added up.

*)
Ym :=	m
		+ p * 0.000376065
		+ in * 0.0254
		+ ft * 0.3048
		+ yd * 0.9144
		+ mile * 1609.344
		+ sm * 1852
		+ fm * 1.829;
Yp := Ym / 0.000376065;
Yin := Ym / 0.0254;
Yft := Ym / 0.3048;
Yyd := Ym / 0.9144;
Ymile := Ym / 1609.344;
Ysm := Ym / 1852;
Yfm := Ym / 1.829;

(*
Länge Meter m SI-Basiseinheit
Astronomische Einheit* AE 1 AE = 149,597 870 · E9 m
Parsec pc 1 pc = 206265 AE = 30,857 · E15 m
Lichtjahr Lj 1 Lj = 9,460 530 · E15 m = 63240 AE = 0,306 59 pc
Ångström Å 1 Å = E–l0 m
typograph. Punkt p 1 p = 0,376 065 mm • im Druckereigewerbe
inch** in 1 in = 2,54 · E–2 m = 25,4 mm***
foot ft 1 ft = 0,3048 m = 30,48 cm
yard yd 1 yd = 0,9144 m
mile mile 1 mile = 1609,344 m
Internat. Seemeile sm 1 sm = 1852 m
Fathom fm 1 fm = 1,829 m • in der Seeschifffahrt

*)
END_FUNCTION_BLOCK

(* POU FINDP, ST *)
FUNCTION FINDP : INT
VAR_INPUT
	str : STRING(STRING_LENGTH);
	src : STRING(STRING_LENGTH);
	pos: INT;
END_VAR
VAR
	i: INT;
	ls: INT;
	lx: INT;
	stp: INT;
END_VAR

(*
version 1.2	29. mar. 2008
programmer 	hugo
tested by	tobias

the function findP searches a string str for the occurence of src beginning at the position pos.

*)
ls := LEN(str);
lx := LEN(src);
IF ls < lx OR lx = 0 THEN RETURN; END_IF;
stp := ls - lx + 1;
FOR i := MAX(pos,1) TO stp DO
	IF MID(str,lx,i) = src THEN
		FINDP := i;
		RETURN;
	END_IF;
END_FOR;
FINDP := 0;

(* revision histroy
hm	4. feb. 2008	rev 1.0
	original release

hm	29. feb 2008	rev 1.1
	ADDED MAX(pos,1) in loop initialization

hm	29. mar. 2008	rev 1.2
	changed STRING to STRING(STRING_LENGTH)
*)	
END_FUNCTION

(* POU FLOAT_TO_REAL, ST *)
FUNCTION FLOAT_TO_REAL : REAL
VAR_INPUT
	FLT : STRING(20);
END_VAR
VAR
	pt : POINTER TO ARRAY[1..20] OF BYTE;
	i: INT;
	X: BYTE;
	sign: INT := 1;
	stop: INT;
	tmp: DINT;
	d : INT;
END_VAR

(*
version 1.3	23. oct. 2008
programmer 	hugo
tested by	oscat

FLOAT_TO_REAL converts a string to a REAL.
the function ignores all wrong characters.
the comma can be , or .
the exponent has to start with capital E or lowercase e .


*)
pt := ADR(FLT);
stop := LEN(FLT);

(* we first check for sign and exit if first number or dot is reached *)
FOR i := 1 TO stop DO
	X := pt^[i];
	IF X > 47 AND X < 58 OR X = 46 THEN
		EXIT;
	ELSIF X = 45 THEN
		(* code 45 is sign *)
		sign := -1;
	END_IF;
END_FOR;

(* now we scan numbers till end or dot or E is reached *)
FOR i := i TO stop DO
	X := pt^[i];
	IF X = 44 OR X = 46 OR X = 69 OR X = 101 THEN
		EXIT;
	(* calculate the value of the digit *)
	ELSIF X > 47 AND x < 58 THEN
		tmp := tmp * 10 + X - 48;
	END_IF;
END_FOR;

(* process the portion after the comma if comma or dot is reached exit if exponent starts *)
IF x = 44 OR X = 46 THEN
	FOR i := i + 1 TO stop DO
		X := pt^[i];
		IF X = 69 OR X = 101 THEN
			EXIT;
		ELSIF x > 47 AND x < 58 THEN
			tmp := tmp * 10 + X - 48;
			d := d - 1;
		END_IF;
	END_FOR;
END_IF;

(* process exponent if present *)
IF X = 69 OR X = 101 THEN
	d := d + DEC_TO_INT(RIGHT(FLT, stop - i));
END_IF;

FLOAT_TO_REAL :=  EXPN(10, d) * DINT_TO_REAL(TMP * SIGN);




(* revision histroy
hm	22. jun. 2008	rev 1.0
	original release

hm	2. oct. 2008	rev 1.1
	fixed an error, characters 8 and 9 would not be converted

hm	22. oct. 2008	rev 1.2
	last fix was not done correctly

hm	23. oct. 2008	rev 1.3
	optimzed code
*)	
END_FUNCTION

(* POU FLOW_CONTROL, ST *)
 FUNCTION_BLOCK FLOW_CONTROL
VAR_INPUT
	IN : BOOL;
	REQ : BOOL;
	ENQ : BOOL;
	RST : BOOL;
END_VAR
VAR_INPUT CONSTANT
	T_AUTO : TIME := T#1h;
	T_DELAY : TIME := T#23h;
END_VAR
VAR_OUTPUT
	Q : BOOL;
	STATUS : BYTE;
END_VAR
VAR
	timer : TP_1D;
END_VAR


(*
version 1.0	28. jun. 2008
programmer 	hugo
tested by	oscat

FLOW_CONTROL switches a valves depending on the input in.
flow control also limits the maximum ontime of the valve and controls pressure on the output side.

*)
STATUS := 100;
IF RST THEN
	Q := FALSE;
	timer(rst := TRUE);
	timer.RST := FALSE;
	STATUS := 103;
ELSIF ENQ THEN
	IF IN THEN
		status := 101;
	END_IF;
	IF REQ THEN
		(* timer will generate a timed pulse after TP goes high *)
		timer.PT1 := T_AUTO;
		timer.PTD := T_DELAY;
		timer.IN := TRUE;
		STATUS := 102;
	END_IF;
END_IF;


(* set output and run timer *)
timer();
timer.IN := FALSE;
Q := (IN AND ENQ) OR timer.Q;



(* revision history
hm 	28. jun. 2008 	rev 1.0
	original version

*)
END_FUNCTION_BLOCK

(* POU FSTRING_TO_BYTE, ST *)
FUNCTION FSTRING_TO_BYTE : BYTE
VAR_INPUT
	IN : STRING(12);
END_VAR
VAR
END_VAR


(*
version 1.1	20. sep. 2008
programmer 	hugo
tested by		oscat

FSTRING_TO_BYTE converts a formatted string into a byte.
the string can be of the form 2#01010, 8#7234, 16#2AD3 and 1234

*)
IF LEFT(IN, 2) = '2#' THEN
	(* we need to convert binary *)
	FSTRING_TO_BYTE := BIN_TO_BYTE(RIGHT(in, LEN(in) - 2));
ELSIF LEFT(in, 2) = '8#' THEN
	(* weneed to convert octals *)
	FSTRING_TO_BYTE := OCT_TO_BYTE(RIGHT(in, LEN(in) - 2));
ELSIF LEFT(in, 3) = '16#' THEN
	(* we need to convert hexadecimal *)
	FSTRING_TO_BYTE := HEX_TO_BYTE(RIGHT(in, LEN(in) - 3));
ELSE
	(* we assume decimal representation *)
	FSTRING_TO_BYTE := DEC_TO_BYTE(CLEAN(in,'0123456789'));
END_IF;


(* revision histroy
hm	18. jun. 2008	rev 1.0
	original release

hm	20. sep. 2008	rev 1.1
	changed length of input string from 20 to 12
*)	
END_FUNCTION

(* POU OCT_TO_BYTE, ST *)
FUNCTION OCT_TO_BYTE : BYTE
VAR_INPUT
	OCT : STRING(10);
END_VAR
VAR
	pt : POINTER TO BYTE;
	i: INT;
	X: BYTE;
	stop: INT;
END_VAR

(*
version 1.1	20. sep. 2008
programmer 	hugo
tested by		oscat

OCT_TO_BYTE converts a octagonal string into a byte.

*)
pt := ADR(oct);
stop := LEN(oct);
FOR I := 1 TO stop DO
	(* read the first character and subtract 48 to get value in decimal 0 = 48 *)
	x := pt^;
	(* calculate the value of the digit *)
	IF X > 47 AND x < 56 THEN
		OCT_TO_BYTE := SHL(OCT_TO_BYTE,3) + X - 48;
	END_IF;
	pt := pt + 1;
END_FOR;



(* revision histroy
hm	18. jun. 2008	rev 1.0
	original release

hm	20. sep. 2008	rev 1.1
	changed length of input string from 20 to 10

*)	
END_FUNCTION

(* POU HEX_TO_BYTE, ST *)
FUNCTION HEX_TO_BYTE : BYTE
VAR_INPUT
	HEX : STRING(5);
END_VAR
VAR
	pt : POINTER TO BYTE;
	i: INT;
	X: BYTE;
	stop: INT;
END_VAR

(*
version 1.1	20. sep. 2008
programmer 	hugo
tested by		oscat

HEX_TO_BYTE converts a Hexadecimal string into a byte.

*)
pt := ADR(hex);
stop := LEN(hex);
FOR I := 1 TO stop DO
	(* read the first character and subtract 48 to get value in decimal 0 = 48 *)
	x := pt^;
	(* calculate the value of the digit *)
	IF X > 47 AND x < 58 THEN
		HEX_TO_BYTE := SHL(HEX_TO_BYTE,4) + X - 48;
	ELSIF X > 64 AND X < 71 THEN
		HEX_TO_BYTE := SHL(HEX_TO_BYTE,4) + X - 55;
	ELSIF X > 96 AND X < 103 THEN
		HEX_TO_BYTE := SHL(HEX_TO_BYTE,4) + X - 87;
	END_IF;
	pt := pt + 1;
END_FOR;




(* revision histroy
hm	18. jun. 2008	rev 1.0
	original release

hm	20. sep.2008	rev 1.1
	changed length of input string from 20 to 5

*)	
END_FUNCTION

(* POU FSTRING_TO_DT, ST *)
FUNCTION FSTRING_TO_DT : DT
VAR_INPUT
	SDT : STRING(60);
	FMT : STRING(60);
END_VAR
VAR CONSTANT
	ignore: STRING(1) := '*';  (* ignore character is * *)
	fchar : STRING(1) := '#';  (* format character is # *)
END_VAR
VAR
	c: STRING(1);
	tmp: STRING(20);
	end: INT;
	dy : INT := 1970;
	dm : INT := 1;
	dd : INT := 1;
	th : INT;
	tm : INT;
	ts : INT;
END_VAR


(*
version 1.0	24. sep. 2008
programmer 	hugo
tested by	oscat

FSTRING_TO_DT converts Formatted String into a DT value.

*)
(* scan input string *)
WHILE fmt <> '' DO
	c := LEFT(fmt,1);
	IF c = ignore THEN
		(* skip ignore characters *)
		fmt := DELETE(fmt,1,1);
		sdt := DELETE(sdt,1,1);
	ELSIF C = fchar THEN
		(* format chracter found skip format char and read identifier *)
		(* store format identifier in c and skip to next char in fmt *)
		c := MID(fmt,1,2);
		fmt := DELETE(fmt,2,1);
		(* extract the substring until the end of sdt or to next char of fmt *)
		IF fmt = '' THEN
			tmp := sdt;
		ELSE
			(* serach for end of substring *)
			end := FIND(sdt, LEFT(fmt,1))-1;
			tmp := LEFT(sdt, end);
			sdt := DELETE(sdt, end,1);
		END_IF;
		(* extract information from substring *)
		IF c = 'Y' THEN
			dy := STRING_TO_INT(tmp);
			IF dy < 100 THEN dy := dy + 2000; END_IF;
		ELSIF c = 'M' THEN
			dm := STRING_TO_INT(tmp);
		ELSIF c = 'N' THEN
			dm := FSTRING_TO_MONTH(tmp,0);
		ELSIF c = 'D' THEN
			dd := STRING_TO_INT(tmp);
		ELSIF c = 'h' THEN
			th := STRING_TO_INT(tmp);
		ELSIF c = 'm' THEN
			tm := STRING_TO_INT(tmp);
		ELSIF c = 's' THEN
			ts := STRING_TO_INT(tmp);
		END_IF;
	ELSIF c = LEFT(sdt,1) THEN
		(* skip matching characters *)
		fmt := DELETE(fmt,1,1);
		sdt := DELETE(sdt,1,1);
	ELSE
		RETURN;
	END_IF;
END_WHILE;

FSTRING_TO_DT := SET_DT(dy,dm,dd,th,tm,ts);


(* revision histroy
hm	24. sep. 2008	rev 1.0
	original release


*)	
END_FUNCTION

(* POU FSTRING_TO_MONTH, ST *)
FUNCTION FSTRING_TO_MONTH : INT
VAR_INPUT
	MTH : STRING(20);
	LANG : INT;
END_VAR
VAR
	lx: INT;
END_VAR


(*
version 1.2	25. oct 2008
programmer 	hugo
tested by	oscat

FSTRING_TO_MONTH converts a string into a month, the string can be a name for the month or a number.
the function is language sensitve when LANG > 1 and checks for all languages when LANG = 0

*)
IF LANG = 0 THEN lx := LANGUAGE.DEFAULT; ELSE lx := MIN(LANG, LANGUAGE.LMAX); END_IF;
MTH := TRIM(mth);
MTH := CAPITALIZE(LOWERCASE(MTH));

FOR FSTRING_TO_MONTH := 1 TO 12 DO
	IF MTH = language.MONTHS[lx, FSTRING_TO_MONTH] THEN RETURN; END_IF;
	IF MTH = language.MONTHS3[lx, FSTRING_TO_MONTH] THEN RETURN; END_IF;
END_FOR;

(* since no name matched try to decode as integer *)
FSTRING_TO_MONTH := STRING_TO_INT(MTH);




(* revision histroy
hm	25. sep. 2008	rev 1.0
	original release

hm	19. oct. 2008	rev 1.1
	changed language setup constants

hm	25. oct. 2008	rev 1.2
	optimized code
*)	
END_FUNCTION

(* POU LOWERCASE, ST *)
FUNCTION LOWERCASE : STRING(STRING_LENGTH)
VAR_INPUT
	str : STRING(STRING_LENGTH);
END_VAR
VAR
	PT : POINTER TO BYTE;
	pos: INT;
	l: INT;
END_VAR

(*
version 1.3	29. mar. 2008
programmer 	hugo
tested by		tobias

lowercase returns str while all letters A..Z and Ä.Ö,Ü are converted to lowercase.

*)
PT := ADR(LOWERCASE);
lowercase := str;
l := LEN(str);
FOR pos := 1 TO l DO
	pt^ := TO_LOWER(pt^);
	PT := PT + 1;
END_FOR;

(* revision histroy
hm	6. oct. 2006	rev 1.0
	original release

hm	4. feb. 2008	rev 1.1
	improved performance
	added Ä.Ö,Ü

hm	6. mar. 2008	rev 1.2
	added support for exteded Ascii

hm	29. mar. 2008	rev 1.3
	changed STRING to STRING(STRING_LENGTH)
*)	
END_FUNCTION

(* POU TO_LOWER, ST *)
FUNCTION TO_LOWER : BYTE
VAR_INPUT
	IN : BYTE;
END_VAR
VAR
END_VAR

(*
version 1.2	25. oct 2008
programmer 	hugo
tested by		tobias

to_lower converts a character from uppercase to lowercase

*)
IF in > 64 AND in < 91 THEN
   TO_LOWER := in OR 16#20;
ELSIF (in > 191 AND in < 223) AND in <> 215 AND setup.EXTENDED_ASCII THEN
   TO_LOWER := in OR 16#20;
ELSE
   TO_LOWER := in;
END_IF;


(* revision history
hm	6. mar. 2008	rev 1.0
	original version

hm	19. oct. 2008	rev 1.1
	changed setup constants

ks	25. oct. 2008	rev 1.2
	optimized code
*)
END_FUNCTION

(* POU FSTRING_TO_DWORD, ST *)
FUNCTION FSTRING_TO_DWORD : DWORD
VAR_INPUT
	IN : STRING(40);
END_VAR
VAR
END_VAR


(*
version 1.1	20. sep. 2008
programmer 	hugo
tested by		oscat

FSTRING_TO_BYTE converts a formatted string into a byte.
the string can be of the form 2#01010, 8#7234, 16#2AD3 and 1234

*)
IF LEFT(IN, 2) = '2#' THEN
	(* we need to convert binary *)
	FSTRING_TO_DWORD := BIN_TO_DWORD(RIGHT(in, LEN(in) - 2));
ELSIF LEFT(in, 2) = '8#' THEN
	(* weneed to convert octals *)
	FSTRING_TO_DWORD := OCT_TO_DWORD(RIGHT(in, LEN(in) - 2));
ELSIF LEFT(in, 3) = '16#' THEN
	(* we need to convert hexadecimal *)
	FSTRING_TO_DWORD := HEX_TO_DWORD(RIGHT(in, LEN(in) - 3));
ELSE
	(* we assume decimal representation *)
	FSTRING_TO_DWORD := DEC_TO_DWORD(CLEAN(in,'0123456789'));
END_IF;


(* revision histroy
hm	18. jun. 2008	rev 1.0
	original release

hm	20. sep. 2008	rev 1.1
	changed length of input dtring from 20 to 40


*)	
END_FUNCTION

(* POU OCT_TO_DWORD, ST *)
FUNCTION OCT_TO_DWORD : DWORD
VAR_INPUT
	OCT : STRING(20);
END_VAR
VAR
	pt : POINTER TO BYTE;
	i: INT;
	X: BYTE;
	stop: INT;
END_VAR

(*
version 1.0	18. jun 2008
programmer 	hugo
tested by	oscat

OCT_TO_DWORD converts a octagonal string into a dword.

*)
pt := ADR(oct);
stop := LEN(oct);
FOR I := 1 TO stop DO
	(* read the first character and subtract 48 to get value in decimal 0 = 48 *)
	x := pt^;
	(* calculate the value of the digit *)
	IF X > 47 AND x < 56 THEN
		OCT_TO_DWORD := SHL(OCT_TO_DWORD,3) + X - 48;
	END_IF;
	pt := pt + 1;
END_FOR;




(* revision histroy
hm	18. jun. 2008	rev 1.0
	original release


*)	
END_FUNCTION

(* POU HEX_TO_DWORD, ST *)
FUNCTION HEX_TO_DWORD : DWORD
VAR_INPUT
	Hex : STRING(20);
END_VAR
VAR
	pt : POINTER TO BYTE;
	i: INT;
	X: BYTE;
	stop: INT;
END_VAR

(*
version 1.4	18. jun. 2008
programmer 	hugo
tested by	tobias

HEX_TO_DWORD converts a Hexadecimal string into a DWORD.

*)
pt := ADR(hex);
stop := LEN(hex);
FOR I := 1 TO stop DO
	(* read the first character and subtract 48 to get value in decimal 0 = 48 *)
	x := pt^;
	(* calculate the value of the digit *)
	IF X > 47 AND x < 58 THEN
		HEX_TO_DWORD := SHL(HEX_TO_DWORD,4) + X - 48;
	ELSIF X > 64 AND X < 71 THEN
		HEX_TO_DWORD := SHL(HEX_TO_DWORD,4) + X - 55;
	ELSIF X > 96 AND X < 103 THEN
		HEX_TO_DWORD := SHL(HEX_TO_DWORD,4) + X - 87;
	END_IF;
	pt := pt + 1;
END_FOR;



(* revision histroy
hm	2.10.2007		rev 1.0
	original release

hm	19.11.2007		rev 1.1
	changed type of function from int to dword

hm 	4. mar 2008		rev 1.2
	added support for a..f and return 0 for invalid string

hm	29. mar. 2008	rev 1.3
	changed STRING to STRING(8)

hm	18. jun. 2008	rev 1.4
	changed input hex to STRING(20)
	function now ignores wrong characters
*)	
END_FUNCTION

(* POU FSTRING_TO_WEEK, ST *)
FUNCTION FSTRING_TO_WEEK : BYTE
VAR_INPUT
	WEEK : STRING(60);
	LANG : INT;
END_VAR
VAR
	pos: INT;
END_VAR


(*
version 1.1	25. oct. 2008
programmer 	hugo
tested by	oscat

FSTRING_TO_WEEK converts a list of weekdays into a byte where each bit represents a day of the week.
bit 6 = mo, 0 = su;

*)
pos := FIND(WEEK, ',');
WHILE pos > 0 DO
	FSTRING_TO_WEEK := FSTRING_TO_WEEK OR SHR(BYTE#128, FSTRING_TO_WEEKDAY(MID(WEEK, pos - 1, 1), LANG));
	WEEK := RIGHT(WEEK, LEN(Week) - pos);
	pos := FIND(WEEK, ',');
END_WHILE;
FSTRING_TO_WEEK := (FSTRING_TO_WEEK OR SHR(BYTE#128, FSTRING_TO_WEEKDAY(WEEK, LANG))) AND BYTE#127;


(* revision histroy
hm	18. jun. 2008	rev 1.0
	original release

hm	25. oct. 2008	rev 1.1
	using language defauls and input lang
*)	
END_FUNCTION

(* POU FSTRING_TO_WEEKDAY, ST *)
FUNCTION FSTRING_TO_WEEKDAY : INT
VAR_INPUT
	WDAY : STRING(20);
	LANG : INT;
END_VAR
VAR
	tmp: STRING(2);
	i: INT;
	ly: INT;
END_VAR


(*
version 1.2	25. oct. 2008
programmer 	hugo
tested by	oscat

FSTRING_TO_WEEKDAY converts a weekday string into an integer 1..7.

*)
IF LANG = 0 THEN ly := LANGUAGE.DEFAULT; ELSE ly := MIN(LANG, LANGUAGE.LMAX); END_IF;
(* tmp needs to be calculated first otherwise find can return wrong values *)
tmp := TRIM(wday);
tmp := CAPITALIZE(LOWERCASE(tmp));
FOR i := 1 TO 7 DO
	IF language.WEEKDAYS2[ly, i] = tmp THEN
		FSTRING_TO_WEEKDAY := i;
		RETURN;
	END_IF;
END_FOR
FSTRING_TO_WEEKDAY := STRING_TO_INT(WDAY);




(* revision histroy
hm	18. jun. 2008	rev 1.0
	original release

hm	18. jul. 2008	rev 1.1
	changed nested call of left(trim()) for compatibility reasons

hm	25. oct. 2008	rev 1.2
	using language constants
*)	
END_FUNCTION

(* POU FT_AVG, ST *)
FUNCTION_BLOCK FT_AVG
VAR_INPUT
	IN : REAL;
	E : BOOL := TRUE;
	N : INT := 32;
	RST : BOOL;
END_VAR
VAR_OUTPUT
	AVG : REAL;
END_VAR
VAR
	buff : DELAY;
	i: INT;
	init : BOOL;
END_VAR

(*
version 1.4	18. oct. 2008
programmer 	hugo
tested by	oscat

this function calculates the moving average over n samples from a sequential input
the input values are shifted into an N deep buffer and the avg of this buffer is diplayed at anytime on the output.
a rst will load the buffer with the current in value..

*)
(* limit n to a max of 32 because delay can do max 32 cycles *)
buff.N := LIMIT(0, N, 32);

IF NOT init OR rst THEN
	FOR i := 1 TO N DO
		buff(in := in);
	END_FOR;
	avg := in;
	init := TRUE;
ELSIF E THEN
	buff(in := in);
	avg := avg + (in - buff.out)/N;
END_IF;

(* revision history

hm	7. jan. 2007	rev 1.1
	chaged rst logic to load the buffer with the actual input value instead of 0.
	added en input to allow better control of signal flow
	added init to load the buffer with in at startup to avoid rampup at beginning.
	deleted unused variable cnt.

hm	14. jun. 2008	rev 1.2
	set default for input en = TRUE and N = 32

hm	10. oct. 2008	rev 1.3
	improved performance

hm	18. oct. 2008	rev 1.4
	changed input en to e for compatibility reasons
	
*)
END_FUNCTION_BLOCK

(* POU FT_IMP, ST *)
FUNCTION_BLOCK FT_IMP
VAR_INPUT
	in : REAL;
	T : TIME;
	K : REAL := 1;
END_VAR
VAR_OUTPUT
	out : REAL;
END_VAR
VAR
	t1 : FT_PT1;
END_VAR

(*
version 1.1	3 Jan 2007
programmer 	hugo
tested by	oscat

FT_IMP is 	an impulse filter (high pass filter) with the time T and factor K.
 
*)
T1(in:= in, T:=T);
out := (in - t1.out) * K;

(*
hm 3.1.2007	rev 1.1
	added factor K

*)
END_FUNCTION_BLOCK

(* POU FT_INT, ST *)
FUNCTION_BLOCK FT_INT
VAR_INPUT
	IN : REAL;
	K : REAL := 1;
	RUN : BOOL := TRUE;
	RST : BOOL;
	OUT_MIN : REAL := -1E37;
	OUT_MAX : REAL := 1E37;
END_VAR
VAR_OUTPUT
	OUT : REAL;
	LIM : BOOL;
END_VAR
VAR
	INTeg : INTEGRATE;
END_VAR


(*
version 2.1	3. nov. 2008
programmer 	hugo
tested by	oscat

FT_int is an integrator with input IN and factor K.
integration is only done while run = true, if run is false integration is stopped and the out remains at the last value.
if run is left unconnected, run is considered true by the function block.
the output ET will display the total integration time from last reset.
the out_min and out_max values can be set to ,imit the output value range. 
the default for K is 1.

 
*)
IF rst THEN
	out := 0;
ELSE
	integ(X := IN, E := RUN, K := K, Y := out);
END_IF;

(* limit the outputs *)
IF out >= OUT_MAX THEN
	out := out_max;
	LIM := TRUE;
ELSIF out <= out_min THEN
	out := out_min;
	lim := TRUE;
ELSE
	lim := FALSE;
END_IF;


(* code with rev 2.0
IF NOT init OR RST THEN
	init := TRUE;
	in_last := in;
END_IF;
CT();
IF rst THEN
	OUT := 0;
	LIM := FALSE;
ELSIF run THEN
	(* call for last cycle time *)
	OUT := (IN + IN_LAST) * 0.5 * CT.TC * K + OUT;
	in_last := in;
END_IF;
(* check output for limits *)
IF OUT > OUT_MAX THEN
	OUT := OUT_MAX;
	LIM := TRUE;
ELSIF OUT < OUT_MIN THEN
	OUT := OUT_MIN;
	LIM := TRUE;
ELSE
	LIM := FALSE;
END_IF;
*)

(*
hm 13.12.2006	rev 1.1
	changed to "trapezregel" which increases accuracy
	before out := out + in * time new: out := out + (in + in_last) / 2 * time

hm 15.1.2007		rev 1.2
	added default for k to be 1.

hm	15.9.2007		rev 1.3
	replaced time() with T_PLC_US for compatibility and performance reason
	increased internal accuracy to microseconds

hm 29. oct 2007		rev 1.4
	changed code so int will not be called is time difference is 0 to increase accuracy on systems
	with cycle times below 1ms

hm	2. dec 2007	 	rev 1.5
	changed code for better performance

hm	5. jan 2008		rev 1.6
	further improvements in performance

hm	8. feb 2008		rev 1.7
	deleted limits +/- 1000 now limit is the range of real
	added variables out1 and out2 to extend the resolution
	corrected an error with elapsed time
	deleted unusfull output ET

hm	13. mar 2008	rev 1.8
	changed preset value out_min to -1e37.
	stop integrator at the limits.

hm	16. mar 2008	rev 1.9
	added type conversion to avoid warning under codesys 3.0

hm	2. jun. 2008	rev 2.0
	rewritten with clear code
	limits can now be set without run

hm	3. nov. 2008	rev 2.1
	optimized code using INTEGRATE and LIMX
*)
END_FUNCTION_BLOCK

(* POU INTEGRATE, ST *)
FUNCTION_BLOCK INTEGRATE
VAR_INPUT
	E : BOOL := TRUE;
	X : REAL;
	K : REAL := 1;
END_VAR
VAR_IN_OUT
	Y : REAL;
END_VAR
VAR
	X_last : REAL;
	init: BOOL;
	last: DWORD;
	tx: DWORD;
END_VAR


(*
version 1.0	3. nov. 2008
programmer 	hugo
tested by	oscat

integrate is a plain integrator with I/O for out.

 
*)
(*read system time *)
tx := T_PLC_MS();

IF NOT init THEN
	init := TRUE;
	X_last := X;
ELSIF E THEN
	Y := (X + X_LAST) * 0.5E-3 * DWORD_TO_REAL(tx-last) * K + Y;
	X_last := X;
END_IF;
last := tx;



(*
hm 	3. nov. 2008	rev 1.0
original version
	
*)
END_FUNCTION_BLOCK

(* POU FT_INT2, ST *)
FUNCTION_BLOCK FT_INT2
VAR_INPUT
	IN : REAL;
	K : REAL := 1;
	RUN : BOOL := 1;
	RST : BOOL;
	OUT_MIN : REAL := -1E37;
	OUT_MAX : REAL := 1E37;
END_VAR
VAR_OUTPUT
	OUT : REAL;
	LIM : BOOL;
END_VAR
VAR
	integ: INTEGRATE;
	ix : REAL;
	val : REAL2;
END_VAR


(*
version 1.1	5. nov. 2008
programmer 	hugo
tested by	oscat

FT_int2 is an integrator with input IN and factor K.
integration is only done while run = true, if run is false integration is stopped and the out remains at the last value.
if run is left unconnected, run is considered true by the function block.
the out_min and out_max values can be set to ,imit the output value range. 
the default for K is 1.
FT_INT2 has double presision accuracy (14 digits).


*)
IF RST THEN
	val := R2_SET(0);
	out := 0;
ELSE
	integ(X := IN, E := RUN, K := K, Y := ix);
	val := R2_ADD(val, ix);
	ix := 0;
	OUT := val.RX;
END_IF;

(* check output for limits *)
IF out > OUT_MIN AND out < OUT_MAX THEN
	LIM := FALSE;
ELSE
	OUT := LIMIT(OUT_MIN, OUT, OUT_MAX);
	val := R2_SET(OUT);
	LIM := TRUE;
END_IF;



(*	revision history
hm	2. jun. 2008	rev 1.0
	original version

hm	5. nov. 2008	rev 1.1
	rewritten code using integrate
*)
END_FUNCTION_BLOCK

(* POU R2_SET, ST *)
FUNCTION R2_SET : REAL2
VAR_INPUT
	X : REAL;
END_VAR
VAR
END_VAR

(*
version 1.0	21. mar. 2008
programmer 	hugo
tested by		tobias

R2_set sets a double precision real to a single real value.

*)
R2_SET.RX := X;
R2_SET.R1 := 0;


(* revision history
hm	2. jun. 2008	rev 1.0
	original version

*)
END_FUNCTION

(* POU FT_MIN_MAX, ST *)
FUNCTION_BLOCK FT_MIN_MAX
VAR_INPUT
	in : REAL;
	rst : BOOL;
END_VAR
VAR_OUTPUT
	mx : REAL;
	mn : REAL;
END_VAR
VAR
	init: BOOL;
END_VAR

(*
version 1.0	1 sep 2006
programmer 	hugo
tested by		tobias

this function block stores the min and max value of an input signal.
when rst is true the mn and mx outputs are set to the in value.
when a rst is never active the function autoresets to the in value at startup.
since the input might not be present at first cycle the mn and mx are set during second cycle.

*)
IF rst OR NOT init THEN
	mn := in;
	mx := in;
	init := 1;
ELSIF in < mn THEN mn := in;
ELSIF in > mx THEN mx := in;
END_IF;
END_FUNCTION_BLOCK

(* POU FT_PD, ST *)
FUNCTION_BLOCK FT_PD
VAR_INPUT
	IN : REAL;
	KP : REAL := 1.0;
	TV : REAL := 1.0;
END_VAR
VAR_OUTPUT
	Y : REAL;
END_VAR
VAR
	diff : FT_DERIV;
END_VAR

(*
version 1.0	3. jun 2008
programmer 	hugo
tested by		tobias

FT_PD is a PD controller.
The PD controller works according to the fomula Y = KP *(IN + DERIV(e) ).

*)
(* run differentiator *)
diff(IN := IN, K := TV);

(* combine both values *)
Y := KP * (diff.out + IN);



(* revision history
hm 	3. jun. 2008 	rev 1.0
	original version


*)
END_FUNCTION_BLOCK

(* POU FT_PDT1, ST *)
FUNCTION_BLOCK FT_PDT1
VAR_INPUT
	IN : REAL;
	KP : REAL := 1.0;
	TV : REAL := 1.0;
	T1 : REAL := 1.0;
END_VAR
VAR_OUTPUT
	Y : REAL;
END_VAR
VAR
	diff : FT_DERIV;
	TP : FT_PT1;
END_VAR

(*
version 1.0	3. jun 2008
programmer 	hugo
tested by		tobias

FT_PD is a PD controller.
The PD controller works according to the fomula Y = KP *(IN + DERIV(e) ).

*)
(* run differentiator *)
diff(IN := IN, K := TV);

(* Run PT1 filter *)
tp(in := diff.out, T := REAL_TO_TIME(T1));

(* combine both values *)
Y := KP * (tp.out + IN);



(* revision history
hm 	3. jun. 2008 	rev 1.0
	original version


*)
END_FUNCTION_BLOCK

(* POU FT_PI, ST *)
FUNCTION_BLOCK FT_PI
VAR_INPUT
	IN : REAL;
	KP : REAL := 1.0;
	KI : REAL := 1.0;
	ILIM_L : REAL := -1E38;
	ILIM_H : REAL := 1E38;
	IEN : BOOL := TRUE;
	RST : BOOL;
END_VAR
VAR_OUTPUT
	Y : REAL;
	LIM : BOOL;
END_VAR
VAR
	integ : FT_INT;
END_VAR

(*
version 2.0	3. jun 2008
programmer 	hugo
tested by		tobias

FT_PI is a PI controller.
The PID controller works according to the fomula Y = IN *(KP+ KI * INTEG(e) ).
a rst will reset the integrator to 0
ilim_h and iLim_l set the possible output range of the internal integrator.
the output flags lim will signal that the output limits are active.

default values for KP = 1, KI = 1, ILIM_L = -1E37, iLIM_H = +1E38.
*)
(* run integrator *)
integ(IN := IN, K := KI, RUN := IEN, RST := RST, OUT_MIN := ILIM_L, OUT_MAX := ILIM_H);

(* check if integrator has reached its limits and set overflow *)
LIM := integ.LIM;
Y := KP * IN + integ.Out;



(* revision history
hm 	3. jun. 2008 	rev 2.0
	original version


*)
END_FUNCTION_BLOCK

(* POU FT_PID, ST *)
FUNCTION_BLOCK FT_PID
VAR_INPUT
	IN : REAL;
	KP : REAL := 1.0;
	TN : REAL := 1.0;
	TV : REAL := 1.0;
	ILIM_L : REAL := -1E38;
	ILIM_H : REAL := 1E38;
	IEN : BOOL := TRUE;
	RST : BOOL;
END_VAR
VAR_OUTPUT
	Y : REAL;
	LIM : BOOL;
END_VAR
VAR
	integ : FT_INT;
	diff : FT_DERIV;
END_VAR

(*
version 2.0	3. jun 2008
programmer 	hugo
tested by		tobias

FT_PI is a PI controller.
The PID controller works according to the fomula Y = IN *(KP+ KI * INTEG(e) ).
a rst will reset the integrator to 0
ilim_h and iLim_l set the possible output range of the internal integrator.
the output flags lim will signal that the output limits are active.

default values for KP = 1, KI = 1, ILIM_L = -1E37, iLIM_H = +1E38.
*)
(* run integrator only if TN > 0 *)
IF TN > 0 THEN
	integ(IN := IN, K := 1 / TN, RUN := IEN, RST := RST, OUT_MIN := ILIM_L, OUT_MAX := ILIM_H);
ELSE
	integ(RST := FALSE);
END_IF;

(* run differentiator *)
diff(IN := IN, K := TV);

(* combine both values *)
Y := KP * (integ.Out + diff.out + IN);

(* check if integrator has reached its limits and set overflow *)
LIM := integ.LIM;



(* revision history
hm 	3. jun. 2008 	rev 2.0
	original version


*)
END_FUNCTION_BLOCK

(* POU FT_PIDW, ST *)
FUNCTION_BLOCK FT_PIDW
VAR_INPUT
	IN : REAL;
	KP : REAL := 1.0;
	TN : REAL := 1.0;
	TV : REAL := 1.0;
	LIM_L : REAL := -1E38;
	LIM_H : REAL := 1E38;
	RST : BOOL;
END_VAR
VAR_OUTPUT
	Y : REAL;
	LIM : BOOL;
END_VAR
VAR
	integ : INTEGRATE;
	diff : FT_DERIV;
	YI: REAL;
END_VAR

(*
version 1.1	5. nov. 2008
programmer 	hugo
tested by	oscat

FT_PIDW is a PID controller with dynamic wind_up reset.
The PID controller works according to the fomula Y = KP *(IN + KI * INTEG(e) + DERIV(e) ).
a rst will reset the integrator to 0
lim_h and Lim_l set the possible output range of the internal integrator.
the output flags lim will signal that the output limits are active.

default values for KP = 1, KI = 1, ILIM_L = -1E37, iLIM_H = +1E38.
*)
(* run the integrator *)
IF tn = 0 OR rst THEN
	integ(E := FALSE, Y := YI);
	YI := 0;
ELSE
	integ(X := IN, K := 1 / TN, E := NOT LIM, Y := YI);
END_IF;

(* add up integrator and linear part *)
Y := KP * (IN + YI);

(* run differentiator *)
diff(IN := IN, K := TV);

(* set lim before differentiator is added to stop integrator if necessary *)
IF Y > LIM_L AND Y < LIM_H THEN
	LIM := FALSE;
ELSE
	LIM := TRUE;
END_IF;

(* add differential part and limit output Y *)

Y := LIMIT(LIM_L, Y + KP * diff.out, LIM_H);




(* revision history
hm 	3. jun. 2008 	rev 1.0
	original version

hm	5. nov. 2008	rev 1.1
	changed code to use integrate
*)
END_FUNCTION_BLOCK

(* POU FT_PIW, ST *)
FUNCTION_BLOCK FT_PIW
VAR_INPUT
	IN : REAL;
	KP : REAL := 1.0;
	KI : REAL := 1.0;
	LIM_L : REAL := -1E38;
	LIM_H : REAL := 1E38;
	RST : BOOL;
END_VAR
VAR_OUTPUT
	Y : REAL;
	LIM : BOOL;
END_VAR
VAR
	integ : FT_INT;
END_VAR

(*
version 1.0	3. jun 2008
programmer 	hugo
tested by		tobias

FT_PIW is a PI controller.
The PID controller works according to the fomula Y = IN *(KP+ KI * INTEG(e) ).
a rst will reset the integrator to 0
ilim_h and iLim_l set the possible output range of the internal integrator.
the output flag lim will signal that the output limits are active.
the controller is equipped with anti wind_up circuitry that stops the integrator when lim_h or lim_l is reached


default values for KP = 1, KI = 1, ILIM_L = -1E37, iLIM_H = +1E38.
*)
(* run integrator *)
integ(IN := IN, K := KI, RUN := NOT LIM, RST := RST);

(* set output value *)
Y := KP * IN + integ.Out;

(* check for limits and set integrator for anti wind up *)
IF Y < LIM_L THEN
	Y := LIM_L;
	LIM := TRUE;
ELSIF Y > LIM_H THEN
	Y := LIM_H;
	LIM := TRUE;
ELSE
	LIM := FALSE;
END_IF;



(* revision history
hm 	3. jun. 2008 	rev 1.0
	original version


*)
END_FUNCTION_BLOCK

(* POU FT_Profile, ST *)
FUNCTION_BLOCK FT_Profile
VAR_INPUT
	K : REAL := 1;
	O : REAL;
	M : REAL := 1;
	E : BOOL;
END_VAR
VAR_INPUT CONSTANT
	value_0 : REAL;
	time_1 : TIME;
	value_1 : REAL;
	time_2 : TIME;
	value_2 : REAL;
	time_3 : TIME;
	value_3 : REAL;
	time_10 : TIME;
	value_10 : REAL;
	time_11 : TIME;
	value_11 : REAL;
	time_12 : TIME;
	value_12 : REAL;
	time_13 : TIME;
	value_13 : REAL;
END_VAR
VAR_OUTPUT
	Y : REAL;
	RUN : BOOL;
	ET : TIME;
END_VAR
VAR
	tx : TIME;
	edge : BOOL;
	state: BYTE;
	ta: TIME;
	tb: TIME;
	t0 : TIME;
	temp: REAL;
	va: REAL;
	vb: REAL;
END_VAR

(*
version 1.1	15 sep 2007
programmer 	tobias
tested by		hugo

FT_Profile generates an output signal which is defined by values over a time scale.
the different values are connected by ramps between the individual values.
a rising edge on E starts the output signal generation and E = True can delay time_3 / value_3 as long as it stays true.
an additional multiplier K can be used to multiply the output and an offset O can be added to the output dynamically.
*)
(* read system time *)
tx := DWORD_TO_TIME(T_PLC_MS());

(* determine start condition *)
IF E AND NOT edge THEN
	RUN := TRUE;
	ET := t#0s;
	t0 := tx;
	ta := tx;
	tb := multime(time_1, M);
	va := value_0;
	vb := value_1;
	temp := value_0;
	state := 1;
END_IF;
edge := E;

(* generate startup profile *)
IF run THEN
	CASE state OF
		1:	IF tx - ta >= tb THEN
				ta := ta + tb;
				tb := multime(time_2 - time_1, M);
				va := value_1;
				vb := value_2;
				temp := value_1;
				state := 2;
			ELSE
				temp := ((vb - va) * TIME_TO_REAL(tx - ta) / TIME_TO_REAL(tb) + va);
			END_IF;
		2:	IF tx - ta >= tb THEN
				ta := ta + tb;
				tb := multime(time_3 - time_2, M);
				va := value_2;
				vb := value_3;
				temp := value_2;
				state := 3;
			ELSE
				temp := ((vb - va) * TIME_TO_REAL(tx - ta) / TIME_TO_REAL(tb) + va);
			END_IF;
		3:	IF tx - ta >= tb THEN
				ta := ta + tb;
				tb := multime(time_10 - time_3, M);
				va := value_3;
				vb := value_10;
				temp := value_3;
				state := 4;
			ELSE
				temp := ((vb - va) * TIME_TO_REAL(tx - ta) / TIME_TO_REAL(tb) + va);
			END_IF;
		4 :	IF tx - ta >= tb THEN
				ta := ta + tb;
				tb := multime(time_11 - time_10, M);
				va := value_10;
				vb := value_11;
				temp := value_10;
				IF E THEN state := 5; ELSE state := 6; END_IF;
			ELSE
				temp := ((vb - va) * TIME_TO_REAL(tx - ta) / TIME_TO_REAL(tb) + va);
			END_IF;
		5:	(* extend the signal while E is true *)
			IF E THEN
				ta := tx;
			ELSE
				state := 6;
			END_IF;
		6:	IF tx - ta >= tb THEN
				ta := ta + tb;
				tb := multime(time_12 - time_11, M);
				va := value_11;
				vb := value_12;
				temp := value_11;
				state := 7;
			ELSE
				temp := ((vb - va) * TIME_TO_REAL(tx - ta) / TIME_TO_REAL(tb) + va);
			END_IF;
		7:	IF tx - ta >= tb THEN
				ta := ta + tb;
				tb := multime(time_13 - time_12, M);
				va := value_12;
				vb := value_13;
				temp := value_12;
				state := 8;
			ELSE
				temp := ((vb - va) * TIME_TO_REAL(tx - ta) / TIME_TO_REAL(tb) + va);
			END_IF;
		8:	IF tx - ta >= tb THEN
				temp := value_13;
				run := FALSE;
			ELSE
				temp := ((vb - va) * TIME_TO_REAL(tx - ta) / TIME_TO_REAL(tb) + va);
			END_IF;
	END_CASE;
	Y := temp * K + O;
	ET := tx - t0;
END_IF;

(* revision history
hm	27 feb 2007		rev 1.0
	original version

hm	15. sep2007		rev 1.1
	replaced Time() with T_PLC_MS for compatibility and performance reasons

*)
END_FUNCTION_BLOCK

(* POU FT_PT2, ST *)
FUNCTION_BLOCK FT_PT2
VAR_INPUT
	in : REAL;
	T : TIME;
	D : REAL;
	K : REAL := 1;
END_VAR
VAR_OUTPUT
	out : REAL;
END_VAR
VAR
	init: BOOL;
	int1 : INTEGRATE;
	int2 : INTEGRATE;
	tn: REAL;
	I1, I2 : REAL;
	tn2: REAL;
END_VAR

(*
version 1.4	3. Nov 2008
programmer 	hugo
tested by	oscat

FT_PT2 is a 2nd grade filter with programmable times T, D and faktor K.
 
*)
(* startup initialisation *)
IF NOT init OR T = T#0s THEN
	init := TRUE;
	out := K * in;
	I2 := out;
ELSE
	TN := TIME_TO_REAL(T) / 1000;
	tn2 := TN * TN;
	int1(X := in * K / TN2 - I1 * 2 * D / TN - I2 / TN2, Y := I1);
	int2(X := I1,Y := I2);
	out := I2;
END_IF;


(* revision history

15.1.2007 hm		rev 1.1
	changed formula to new more acurate formula
	old code:
	tx := TIME();
	IF NOT init THEN
		last := tx;
		init := TRUE;
	ELSE
		IF T> t#0s THEN
			out1 := out1 + (in - out1) * TIME_TO_REAL(Tx - last) / TIME_TO_REAL(T);
		ELSE
			out1 := in;
		END_IF;
		IF T > t#0s THEN
			out2 := out2 + (out1 - out2) * TIME_TO_REAL(Tx - last) / TIME_TO_REAL(T);
		ELSE
			out2 := out1;
		END_IF;
		out := out2 * K;
	END_IF;
	last := tx;


hm 		15.9.2007		rev 1.2
	deleted unused code for init system time reading tx	

hm		30.11.2007		rev 1.3
	changed out to be K * in during initialization
	avoind divide by 0 if tn = 0

hm	3. nov. 2008	rev 1.4
	optimized code and fixed a problem with init
*)
END_FUNCTION_BLOCK

(* POU FT_TN16, ST *)
FUNCTION_BLOCK FT_TN16
VAR_INPUT
	in : REAL;
	T : TIME;
END_VAR
VAR_OUTPUT
	out : REAL;
	trig : BOOL;
END_VAR
VAR
	length : INT := 16;
	X : ARRAY[0..15] OF REAL;
	cnt : INT;
	last : TIME;
	tx: TIME;
	init: BOOL;
END_VAR

(*
version 1.1	16 sep 2007
programmer 	hugo
tested by		tobias

FT_TN16 is delay function, it will delay a signal by a specified time : T and will store 16 values of in before they are put thru to out.
for higher or lower resolution please use FT_TN8 or FT_TN64 instead.
 
*)
(* read system time *)
tx := DWORD_TO_TIME(T_PLC_MS());

trig := FALSE;
IF NOT init THEN
	x[cnt] := in;
	init := TRUE;
	last := tx;
ELSIF tx - last >= T / length THEN
	IF cnt = length - 1 THEN cnt := 0; ELSE cnt := cnt + 1; END_IF;
	Out := X[cnt];
	x[cnt] := in;
	last := tx;
	Trig := TRUE;
END_IF;

(* revision history
hm		1. jan 2007		rev 1.0
	original version

hm		16. sep 2007	rev 1.1
	changes time() to T_plc_ms() for compatibility reasons

*)
END_FUNCTION_BLOCK

(* POU FT_TN64, ST *)
FUNCTION_BLOCK FT_TN64
VAR_INPUT
	in : REAL;
	T : TIME;
END_VAR
VAR_OUTPUT
	out : REAL;
	trig: BOOL;
END_VAR
VAR
	length : INT := 64;
	X : ARRAY[0..63] OF REAL;
	cnt : INT;
	last : TIME;
	tx: TIME;
	init: BOOL;
END_VAR

(*
version 1.1	15 sep 2007
programmer 	hugo
tested by		tobias

FT_TN7 is delay function, it will delay a signal by a specified time : T and will store 64 values of in before they are put thru to out.
if lower resolution is needed, pls use FT_TN8 or FT_TN16 instead.
 
*)
(* read system time *)
tx := DWORD_TO_TIME(T_PLC_MS());

trig := FALSE;
IF NOT init THEN
	x[cnt] := in;
	init := TRUE;
	last := tx;
ELSIF tx - last >= T / length THEN
	IF cnt = length - 1 THEN cnt := 0; ELSE cnt := cnt + 1; END_IF;
	Out := X[cnt];
	x[cnt] := in;
	last := tx;
	trig := TRUE;
END_IF;

(* revision history
hm		1. jan 2007		rev 1.0
	original version

hm		16. sep 2007	rev 1.1
	changes time() to T_plc_ms() for compatibility reasons

*)
END_FUNCTION_BLOCK

(* POU FT_TN8, ST *)
FUNCTION_BLOCK FT_TN8
VAR_INPUT
	in : REAL;
	T : TIME;
END_VAR
VAR_OUTPUT
	out : REAL;
	trig: BOOL;
END_VAR
VAR
	length : INT := 8;
	X : ARRAY[0..7] OF REAL;
	cnt : INT;
	last : TIME;
	tx: TIME;
	init: BOOL;
END_VAR

(*
version 1.1	15 Sep 2007
programmer 	hugo
tested by		tobias

FT_TN8 is delay function, it will delay a signal by a specified time : T and will store 8 values of in before they are put thru to out.
if higher resolution is needed, pls use FT_TN16 or FT_TN64 instead.
 
*)
tx := DWORD_TO_TIME(T_PLC_MS());
trig := FALSE;
IF NOT init THEN
	x[cnt] := in;
	init := TRUE;
	last := tx;
ELSIF tx - last >= T / length THEN
	IF cnt = length - 1 THEN cnt := 0; ELSE cnt := cnt + 1; END_IF;
	Out := X[cnt];
	x[cnt] := in;
	last := tx;
	trig := TRUE;
END_IF;

(* revision history
hm		1. jan 2007		rev 1.0
	original version

hm		16. sep 2007	rev 1.1
	changes time() to T_plc_ms() for compatibility reasons

*)
END_FUNCTION_BLOCK

(* POU GAUSS, ST *)
FUNCTION GAUSS : REAL
VAR_INPUT
	X : REAL;
	U : REAL;
	SI: REAL;
END_VAR
VAR
	temp: REAL;
	si_inv: REAL;
END_VAR


(*
version 1.1	27. oct. 2008
programmer 	hugo
tested by	tobias

this function calculates the gaussian density function

*)
temp := X-U;
si_inv := 1 / si;
GAUSS := EXP(Temp * Temp * si_inv * SI_inv * -0.5) * 0.39894228 * si_inv;



(* revision hisdtory
hm	6. apr. 2008	rev 1.0
	original version

hm	27. oct. 2008	rev 1.1
	optimized performance	

*)
END_FUNCTION

(* POU GAUSSCD, ST *)
FUNCTION GAUSSCD : REAL
VAR_INPUT
	X : REAL;
	U : REAL;
	SI: REAL;
END_VAR
VAR
END_VAR


(*
version 1.0	6. apr. 2008
programmer 	hugo
tested by	tobias

this function calculates the gaussian cumulative distribution function

*)
GAUSSCD := (ERF((X - U)/(SI * 1.414213562)) + 1) * 0.5;



(* revision hisdtory
hm	6. apr. 2008	rev 1.0
	original version

*)
END_FUNCTION

(* POU GDF, ST *)
FUNCTION GDF : REAL
VAR_INPUT
	X : REAL;
END_VAR
VAR
END_VAR


(*
version 1.1	18. oct. 2008
programmer 	hugo
tested by	tobias

this function calculates the Gudermannian function.

*)
IF X = 0 THEN
	GDF := 0;
ELSIF X > 15 THEN
	GDF := math.PI05;
ELSIF X < -15 THEN
	GDF := -math.PI05;
ELSE
	GDF := ATAN(EXP(X)) * 2 - math.PI05;
END_IF;

(* revision history
hm	27. apr. 2008	rev 1.0
	original version

hm	18. oct. 2008	rev 1.1
	using math constants
*)
END_FUNCTION

(* POU GEN_BIT, ST *)
FUNCTION_BLOCK GEN_BIT
VAR_INPUT
	in0 : DWORD;
	in1 : DWORD;
	in2 : DWORD;
	in3 : DWORD;
	clk : BOOL;
	steps : INT;
	rep : INT;
	rst : BOOL;
END_VAR
VAR_OUTPUT
	Q0 :BOOL;
	Q1 :BOOL;
	Q2 :BOOL;
	Q3 :BOOL;
	cnt : INT;
	run : BOOL;
END_VAR
VAR
	r0: DWORD;
	r1: DWORD;
	r2: DWORD;
	r3: DWORD;
	rx : INT := 1;
END_VAR

(*
version 1.1	15. oct 2008
programmer 	hugo
tested by		tobias

gen_bit is 4 bit sequencial pattern generator with 4 DWORD inputs and 4 serial outputs.
with the first clock pulse after a reset or after power on, bit 0 of the input DWORDS IN is present on the Outputs Q and the next clock cycle shifts to Bit 1 and so on.
the input steps defines how many bits of the input dwords will be shifted to the outputs. the sequence can be repetive when rep = 0 or any amount of repetitions can be defined with input rep.

*)
(* check if number of runs is finished or rep = 0 which means continuous *)

IF clk AND NOT rst THEN
	run := (rep = 0) OR (rx <= rep);
	IF run THEN
		(* check for step counter reached and reset to 0 if cnt = steps *)
		IF cnt = steps THEN
			cnt := 0;
		END_IF;

		(* when cnt = 0 then reload the inputs into the registers *)
		IF cnt = 0 THEN
			r0 := in0;
			r1 := in1;
			r2 := in2;
			r3 := in3;
		END_IF;

		(* when cnt < steps, shift the lowest bits to the outputs *)
		IF (cnt < steps) THEN
			Q0 := r0.0;
			Q1 := r1.0;
			Q2 := r2.0;
			Q3 := r3.0;
			r0 := SHR(r0,1);
			r1 := SHR(r1,1);
			r2 := SHR(r2,1);
			r3 := SHR(r3,1);
		END_IF;

		(* increment the step counter *)
		cnt := cnt +1;
		IF (cnt = steps) AND (rep <> 0) THEN rx := rx +1; END_IF;
		IF (rx > rep) AND (rep <> 0) THEN run := FALSE; END_IF;
	END_IF;
ELSE
	IF rst THEN
		run := Q0 := Q1 := Q2 := Q3 := FALSE;
		r0 := r1 := r2 := r3 := 0;
		cnt := 0;
		rx := 1;
	END_IF;
END_IF;



(* revision histroy
hm	4 aug 2006	rev 1.0
	original version

hm 15. oct. 2008	rev 1.1
	improved performance



*)
END_FUNCTION_BLOCK

(* POU GEN_PW2, ST *)
FUNCTION_BLOCK GEN_PW2
VAR_INPUT
	ENQ : BOOL;
	TH1 : TIME;
	TL1 : TIME;
	TH2 : TIME;
	TL2 : TIME;
	TS : BOOL;
END_VAR
VAR_OUTPUT
	Q : BOOL;
	TH : TIME;
	TL : TIME;
END_VAR
VAR
	t_high : TIME;
	t_low : TIME;
	tx : TIME;
	start : TIME;
	init : BOOL;
	et : TIME;
END_VAR

(*
version 1.0	26. sep. 2008
programmer 	hugo
tested by	oscat

GEN_PW2 generates a time TH? followed by a time TL?.
the input ts selects between 2 sets of timings for the operation.


*)
(* read system timer *)
tx := DWORD_TO_TIME(T_PLC_MS());

(* startup initialization *)
IF NOT init THEN
	start := tx;
	init := TRUE;
	TH := TL := T#0s;
END_IF;

(* timing selection *)
IF TS THEN
	t_high := TH2;
	t_low := TL2;
ELSE
	t_high := TH1;
	t_low := TL1;
END_IF;

(* normal operation *)
IF ENQ THEN
	et := tx - start;
	IF NOT Q THEN
		IF et >= t_low THEN
			Q := TRUE;
			start := tx;
			TL := T#0s;
		ELSE
			TL := et;
		END_IF;
	ELSE
		IF et >= t_high THEN
			Q := FALSE;
			start := tx;
			TH := T#0s;
		ELSE
			TH := et;
		END_IF;
	END_IF;
ELSE
	Q := FALSE;
	TH := TL := T#0s;
	start := tx;
END_IF



(* revision history
hm		26. sep. 2008		rev 1.0
	original version


*)
END_FUNCTION_BLOCK

(* POU GEN_RDM, ST *)
FUNCTION_BLOCK GEN_RDM
VAR_INPUT
	PT : TIME;
	AM : REAL := 1;
	OS : REAL;
END_VAR
VAR_OUTPUT
	Q : BOOL;
	Out : REAL;
END_VAR
VAR
	tx : TIME;
	last : TIME;
	init : BOOL;
END_VAR

(*
	version 1.1	16 sep 2007
	programmer 	oscat
	tested BY		oscat

this signal generator generates a random output. The signal is defined by period time (PT), 
amplitude (AM), offset (OS).
The Output waveform will have its max peak at AM/2 + OS and its minimum peak at -AM/2 + OS. 
The period time PT defines how often the output signal will jump to a new randow value.
The Output Q will be true for one cycle anytime the output OUT has changed

*)
(* read system time and prepare input data *)
tx := DWORD_TO_TIME(T_PLC_MS()) - last;

(* init section *)
IF NOT init THEN
	init := TRUE;
	last := tx;
	tx := t#0s;
END_IF;

(* add last if one cycle is finished *)
IF tx >= pt THEN
	last := last + pt;
	tx := tx - pt;

	(* generate output signal *)
	out := am * (RDM(0) - 0.5) + os;
	q := TRUE;
ELSE
	q := FALSE;
END_IF;

(* revision history

hm	7.2.2007		rev 1.0
	original version

hm	16.9.2007		rev 1.1
	changes time() to T_plc_ms() for compatibility reasons

*)
END_FUNCTION_BLOCK

(* POU GEN_RDT, ST *)
FUNCTION_BLOCK GEN_RDT

VAR_INPUT
	Enable		 : BOOL := TRUE ;
	Min_Time_ms	: TIME := t#1s ; (* min Taktzeit *)
	Max_Time_ms	: TIME := t#1.2s ; (* Max Taktzeit *)
	TP_Q		 : TIME := t#100ms ; (* Zeit Ausgang auf TRUE *)
END_VAR
VAR_OUTPUT
	xQ		 : BOOL ;
END_VAR
VAR
	(* Taktgenerator Simulation *)
	tonRDMTimer	: TON ; (* Zeitbaustein Taktgenerator *)
	tof_xQ		: TOF ; (* Ausschaltverzögerung Taktgenerator *)
	tRDMTime	: TIME ; (* Sollzeit *)
	rRDMTime	: REAL ; (* Zufalswert Timer *)
END_VAR

(*
version 1.1	16 mar. 2008
programmer 	J. Schohaus
tested by	Hugo

RDMT generates a defined pulse with pulse width TP_Q at random times. the random time will be defined with an minimum and maximum time.

*)


(*
FUNCTION_BLOCK RDMTimer
###############################################################################
		 Ersteller / author :		 		 		 		 		 J.Schohaus
		 Datum / date:		 		 		 		 		 		 13.07.2007
###############################################################################
		 Änderungen / Datum / Ersteller :		 		 		 		 		 		 		 		 		 		 		 		 		 		 		 
		 moditication / date / author :		 		 
###############################################################################
		 Verwendete Bibliotheken		 ( * werden im Baustein nicht benötigt )
		 		 		 		 Oscat.lib
###############################################################################
Beschreibung:
*)
tonRDMTimer ( IN:= Enable , PT:= tRDMTime );
tof_xQ ( IN:= tonRDMTimer.Q , PT:= TP_Q );
XQ := tof_xq.Q;
IF tonRDMTimer.Q THEN
		 xQ := TRUE ;
		 rRDMTime := RDM ( last:= rRDMTime ) ;
		 tRDMTime := REAL_TO_TIME ( rRDMTime * DINT_TO_REAL(TIME_TO_DINT( Max_Time_ms - Min_Time_ms ) + TIME_TO_DINT(Min_Time_ms ))) ;
		 tonRDMTimer ( IN:= FALSE );
END_IF;

(* revision history
J. Schohaus	19. nov 2007	rev 1.0
	origial version

hm	16. mar. 2008			rev 1.1
	added type conversion to avoid warnings under codesys 3.0
*)
END_FUNCTION_BLOCK

(* POU GEN_RMP, ST *)
FUNCTION_BLOCK GEN_RMP
VAR_INPUT
	PT : TIME := t#1s;
	AM : REAL := 1;
	OS : REAL;
	DL : REAL;
END_VAR
VAR_OUTPUT
	Q : BOOL;
	OUT : REAL;
END_VAR
VAR
	tx : TIME;
	last : TIME;
	init : BOOL;
	temp : REAL;
	ltemp: REAL;
END_VAR

(*
	version 1.3	26. oct. 2008
	programmer 	oscat
	tested BY		oscat

this signal generator generates a ramp wave output. The ramp wave signal is defined by period time (PT), 
amplitude (AM), offset (OS) and a specific delay for the output signal (DL).
The Output waveform will have its minimum peak at OS and its maximum peak at AM + OS. 
The delay input can delay a signal up to PT, this can be useful to synchronize different generators 
and generate interleaving signals.
in addition to the analog output Out there is a second boolean output Q with is true for one cycle when the ramp starts.
*)
(* read system time and prepare input data *)
tx := DWORD_TO_TIME(T_PLC_MS()) - last;
DL := modR(dl,1);
IF dl < 0 THEN dl := 1 - dl; END_IF;

(* init section *)
IF NOT init THEN
	init := TRUE;
	last := tx;
	tx := t#0s;
END_IF;

(* add last if one cycle is finished *)
IF tx >= pt THEN
	last := last + pt;
	tx := tx - pt;
END_IF;

(* generate sine wave *)
ltemp := temp;
IF pt > t#0s THEN temp := fract(TIME_TO_REAL(tx + multime(pt, dl)) / TIME_TO_REAL(pt)); END_IF;
out := am * temp + os;

(* boolean output Q *)
Q := temp < ltemp;

(* revision history
hm	3. mar 2007		rev 1.0
	original version

hm	17 sep 2007		rev 1.1
	replaced time() with t_plc_ms for compatibilitx reasons

hm	27. nov 2007	rev 1.2
	avoid divide by 0 when pt = 0

ks	26. oct. 2008	rev 1.3
	code optimization
*)
END_FUNCTION_BLOCK

(* POU GEN_SIN, ST *)
FUNCTION_BLOCK GEN_SIN
VAR_INPUT
	PT : TIME;
	AM : REAL := 1;
	OS : REAL;
	DL : REAL;
END_VAR
VAR_OUTPUT
	Q : BOOL;
	Out : REAL;
END_VAR
VAR
	tx : TIME;
	last : TIME;
	init : BOOL;
	temp : REAL;
END_VAR

(*
version 1.5	18. oct. 2008
programmer 	oscat
tested BY	oscat

this signal generator generates a sine wave output. The sine wave signal is defined by period time (PT), 
amplitude (AM), offset (OS) and a specific delay for the output signal (DL).
The Output waveform will have its max peak at AM/2 + OS and its minimum peak at -AM/2 + OS. 
The delay input can delay a signal up to PT, this can be useful to synchronize different generators 
and generate interleaving signals. A Cos wave can be generated accordingly.
in addition to a analog output Out there is a second boolean output Q with the corresponding binary signal.
*)
(* read system time and prepare input data *)
tx := DWORD_TO_TIME(T_PLC_MS()) - last;
DL := modR(dl,1);
IF dl < 0 THEN dl := 1 - dl; END_IF;

(* init section *)
IF NOT init THEN
	init := TRUE;
	last := tx;
	tx := t#0s;
END_IF;

(* add last if one cycle is finished *)
IF tx >= pt THEN
	last := last + pt;
	tx := tx - pt;
END_IF;

(* generate sine wave *)
IF pt > t#0s THEN temp := SIN(math.PI2 * DWORD_TO_REAL(TIME_TO_DWORD(tx + MULTIME(pt, dl))) / DWORD_TO_REAL(TIME_TO_DWORD(pt))); END_IF;
out := am * 0.5 *  temp + os;

(* boolean output Q *)
q := NOT SIGN_R(temp);

(* revision history
hm	22. jan 2007	rev 1.0
	original version

hm	17 sep 2007	rev 1.1
	replaced time() with t_plc_ms for compatibilitx reasons

hm	27. nov 2007	rev 1.2
	avoid divide by 0 when pt = 0

hm	6. jan 2008		rev 1.3
	improved performance

hm	16. mar. 2008	rev 1.4
	added type conversion to avoid warnings under codesys 3.0

hm	18. oct. 2008	rev 1.5
	using math constants
*)
END_FUNCTION_BLOCK

(* POU GEN_SQ, ST *)
FUNCTION_BLOCK GEN_SQ
VAR_INPUT
	PT : TIME;
END_VAR
VAR_OUTPUT
	Q : BOOL;
END_VAR
VAR
	pti : TIME;
	run: BOOL;
	next_edge: TIME;
	overflow: BOOL;
	tx: TIME;
END_VAR

(*
version 1.1	17 sep 2007
programmer 	hugo
tested by		tobias

gen_sq generates square wave signal with programmable period time.
the period time is defined for 10ms .. 65s
if the period time is set to less then 10ms the min perid is 10ms.

*)
(* read system time *)
tx := DWORD_TO_TIME(T_PLC_MS());

IF NOT run THEN
	next_edge := Tx;
	run := TRUE;
	IF pt < T#10ms THEN PTI := T#5ms; ELSE pti := pt / 2; END_IF;
END_IF;
IF (Tx >= next_edge) AND NOT overflow THEN
	Q := NOT Q;
	IF next_edge + pti < next_edge THEN
		(* time() will overflow every 50 days *)
		overflow := TRUE;
	END_IF;
	next_edge := next_edge + pti;
ELSE
	(* wait till time() has an overflow and reset overflow *)
	IF Tx <= next_edge THEN overflow := FALSE; END_IF;
END_IF;

(* revision history
hm	4. aug 2006		rev 1.0
	original version

hm	17. sep 2007	rev 1.1
	replaced time() with T_PLC_MS() for compatibility reasons

*)
END_FUNCTION_BLOCK

(* POU GEN_SQR, ST *)
FUNCTION_BLOCK GEN_SQR
VAR_INPUT
	PT : TIME;
	AM : REAL;
	OS : REAL;
	DC : REAL := 0.5;
	DL : REAL;
END_VAR
VAR_OUTPUT
	Q : BOOL;
	Out : REAL;
END_VAR
VAR
	tx : TIME;
	last : TIME;
	init: BOOL;
END_VAR

(*
	version 1.3	6. jan 2008
	programmer 	oscat
	tested BY		oscat

this signal generator generates a square wave output. The square wave signal is defined by period time (PT), 
amplitude (AM), offset (OS), duty cycle (DC) and a specific delay for the output signal (DL).
The Output waveform will switch between AM/2 + OS and -AM/2 + OS. The DC input specifies ther duty cycle, 
DC = 0 means output is low at all times and 1 means output is high at all times.
The delay input can delay a signal up to PT, this can be useful to synchronize different generators and generate interleaving signals.
in addition to a analog output Out there is a second boolean output Q.
*)
(* check dc = 1 or 0 *)
IF dc = 0 THEN
	out := -am * 0.5 + os;
	Q := FALSE;
	RETURN;
ELSIF dc = 1 THEN
	out := am * 0.5 + os;
	Q := TRUE;
	RETURN;
END_IF;

(* read system time and prepare input data *)
tx := DWORD_TO_TIME(T_PLC_MS()) - last;
DL := modR(dl,1);
IF dl < 0 THEN dl := 1 - dl; END_IF;
dc := modR(dc,1);
IF dc < 0 THEN dc := 1 - dc; END_IF;

(* init section *)
IF NOT init THEN
	init := TRUE;
	last := tx;
	tx := t#0s;
END_IF;

(* add last if one cycle is finished *)
IF tx >= pt THEN
	last := last + pt;
	tx := tx - pt;
END_IF;

(* check if falling or rising edge first *)
IF multime(pt, dl + dc) >= pt THEN
	(* generate falling edge *)
	IF tx >= multime(pt, dl + dc - 1) THEN
		out := -am * 0.5 + os;
		Q := FALSE;
	END_IF;
	(* generate rising edge *)
	IF tx >= multime(pt, dl) THEN
		out := am * 0.5 + os;
		Q := TRUE;
	END_IF;
ELSE
	(* generate rising edge first *)
	IF tx >= multime(pt, dl) THEN
		out := am * 0.5 + os;
		Q := TRUE;
	END_IF;
	(* generate falling edge *)
	IF tx >= multime(pt, dl + dc) THEN
		out := -am * 0.5 +os;
		Q := FALSE;
	END_IF;
END_IF;

(* revision history

hm	12. feb 2007	rev 1.1
	added default value for dc = 0.5

hm	17 sep 2007		rev 1.2
	replaced time() with t_plc_ms for compatibilitx reasons

hm	6. jan 2008		rev 1.3
	improved performance
*)
END_FUNCTION_BLOCK

(* POU GOLD, ST *)
FUNCTION GOLD : REAL
VAR_INPUT
	X : REAL;
END_VAR
VAR
END_VAR


(*
version 1.0	27. apr. 2008
programmer 	hugo
tested by	tobias

this function calculates the golden function.

*)
GOLD := (X + SQRT(X*X + 4)) * 0.5;


(* revision history
hm	27. apr. 2008	rev 1.0
	original version

*)
END_FUNCTION

(* POU HEAT_INDEX, ST *)
FUNCTION HEAT_INDEX : REAL
VAR_INPUT
	T : REAL;
	RH : REAL;
END_VAR
VAR
	RH2 : REAL;
	T2 : REAL;
END_VAR

(*
version 1.2	2 dec 2007
programmer 	hugo
tested by		tobias

this function calculates the heat index temperature depending on external temperature and Relative humidity

*)
IF RH < 20 OR T < 20 THEN
	Heat_index := T;
ELSE
	RH2 := RH * RH;
	T := C_to_F(T);
	T2 := T * T;
	Heat_index := -42.379 + 2.04901523 * T - 6.83783E-3 * T2
			+ RH * (10.1433127 - 0.22475541 * T + 1.22874E-3 * T2)
			+ RH2 * (8.5282E-4 * T - 5.481717E-2 - 1.99E-6 * T2);
	Heat_index := F_to_C(Heat_index);
END_IF;

(* revision history

hm 27.2.2007		rev 1.1
	deleted unused variables rh3 and T3

hm	2.12.2007		rev 1.2
	changed code for better performance
*)
END_FUNCTION

(* POU HEAT_METER, ST *)
FUNCTION_BLOCK HEAT_METER
VAR_INPUT
	TF, TR : REAL;
	LPH : REAL;
	E : BOOL;
	RST : BOOL;
END_VAR
VAR_INPUT CONSTANT
	CP : REAL;
	Density : REAL;
	Content : REAL;
	Pulse_Mode : BOOL;
	Return_meter : BOOL;
	AVG_time : TIME := T#5s;
END_VAR
VAR_OUTPUT
	Y : REAL;
	C : REAL;
END_VAR
VAR
	tx, last : DWORD;
	int1 : FT_INT2;
	edge : BOOL;
	X: REAL;
	init: BOOL;
	Y_last: REAL;
END_VAR

(*
version 1.5	6. nov. 2008
programmer 	hugo
tested by	oscat

Heat meter measures the heat transfer of water of a mixture of water and another component.
The inputs are foreward temperature and reverse temperature.
the additional component is specified with its parameters density, Specific heat capacity and content in %.
an input e anables the measurement while it can be configured to be based on X liters / pulse or in liters / hour.
the output is in Joule.

*)
IF rst THEN
	int1(rst := TRUE);
	int1.rst := FALSE;
	C := Y := 0;
ELSIF e THEN
	X := (WATER_DENSITY(SEL(return_meter, TF, TR), FALSE) * (WATER_ENTHALPY(TF) - WATER_ENTHALPY(TR)) * (1-content) + CP * Density * content*(TF-TR));
	IF pulse_mode THEN
		IF NOT edge THEN Y := Y + X * LPH; END_IF;
	ELSE
		int1(in := X * LPH / 3600.0, out_min := 0, out_max := 3E38);
		Y := int1.Out;
	END_IF;
END_IF;

(* store the value of e *)
edge := e;

(* read system_time *)
tx := T_PLC_MS();

(* only init at startup necessary *)
IF NOT init THEN
	init := TRUE;
	last := tx;
END_IF;

(* calculate the current consumption *)
IF (tx - last >= TIME_TO_DWORD(AVG_TIME)) AND (avg_time > T#0s) THEN
	last := tx;
	C := (Y - Y_last) * 3.6/DWORD_TO_REAL(TIME_TO_DWORD(AVG_TIME));
	Y_last := Y;
END_IF;



(* revision history
hm	16. nov. 2007	rev 1.0
	original version

hm	24. dec. 2007	rev 1.1
	added config variable return_meter
	added output C for current consumption

hm	6. mar. 2008	rev 1.2
	corrected an error in pulse mode

hm	16. mar. 2008	rev 1.3
	added type conversion to avoid warnings under codesys 3.0

hm	21. oct. 2008	rev 1.4
	improved code

hm	6. nov. 2008	REV 1.5
	changed to FT_INT2 to avoid overrun at hig values
*)
END_FUNCTION_BLOCK

(* POU WATER_DENSITY, ST *)
FUNCTION WATER_DENSITY : REAL
VAR_INPUT
	T : REAL;
	Sat : BOOL;
END_VAR
VAR CONSTANT
	a0 : REAL := 999.83952;
	a1 : REAL := 16.952577;
	a2 : REAL := -7.9905127E-3;
	a3 : REAL := -4.6241757E-5;
	a4 : REAL := 1.0584601E-7;
	a5 : REAL := -2.8103006E-10;
	b  : REAL := 0.0168872;
END_VAR
VAR
	T2: REAL;
	T4: REAL;
END_VAR


(*
version 1.1	2 dec 2007
programmer 	hugo
tested by		tobias

this function calculates the water density for air free water between 0 and 100 deg C
while sat is false the denisty is calculated for air free water and when sat = true
the calculation is performed for water saturated with air.

*)
T2 := T * T;
T4 := T2 * T2;

(* original code changed for performance
Water_density := (a0 + a1*T + a2*EXPT(T,2) + a3*EXPT(t,3) + a4*EXPT(t,4) + a5*EXPT(t,5)) / (1 + b*T);
*)
Water_density := (a0 + a1*T + a2*T2 + a3*T2*T + a4*T4 + a5*T4*T) / (1 + b*T);

IF sat THEN Water_density := Water_density - 0.004612 + 0.000106 * T; END_IF;


(* revision history

hm	13.9.2007		rev 1.0
	original version

hm	2.12.2007		rev 1.1
	changed code for better performance
*)

(*
    °C - die Celsius-Temperatur in Grad Celsius
    v – das spezifische Volumen in Kubikdezimeter je Kilogramm dm³/kg
    h – die spezifische Enthalpie in Kilojoule je Kilogramm 	kJ/kg
    u – die spezifische Innere Energie in Kilojoule je Kilogramm 	kJ/kg
    s – die spezifische Entropie in Kilojoule je Kilogramm mal Kelvin 	kJ/(kg·K)
    cp - die spezifische Wärmekapazität bei konstantem Druck in Kilojoule je Kilogramm mal Kelvin 	kJ/(kg·K)
    Y – Volumenausdehnungskoeffizient in 10-3 durch Kelvin  10-3/K
    L – Wärmeleitfähigkeit in Milliwatt je Meter mal Kelvin  mW / (m·K) 
    n – Viskosität in Mikropascal mal Sekunde uPa·s 	
    s ? – Oberflächenspannung in Millinewton je Meter  mN/m


°C 		v 				h 			u 		s 			cp 		Y 		L		n		s	
-20		1,006580	
0 		1,000160 		0,06 		-0,04 	-0,0001 	4,228 	-0,080 	561,0 	1792 	75,65
4		1,000028
5 		1,0000 		21,1 		21,0 	0,076 		4,200 	0,011 	570,6 	1518 	74,95
10 		1,0003 		42,1 		42,0 	0,151 		4,188 	0,087 	580,0 	1306 	74,22
15 		1,0009 		63,0 		62,9 	0,224 		4,184 	0,152 	589,4 	1137 	73,49
20 		1,001797 		83,9 		83,8 	0,296 		4,183 	0,209 	598,4 	1001 	72,74
25 		1,0029 		104,8 		104,7 	0,367 		4,183 	0,259 	607,2 	890,4 	71,98
30 		1,0044 		125,8 		125,7 	0,437 		4,183 	0,305 	615,5 	797,7 	71,20
35 		1,0060 		146,7 		146,6 	0,505 		4,183 	0,347 	623,3 	719,6 	70,41
40 		1,007842 		167,58 	167,5 	0,572 		4,182 	0,386 	630,6 	653,3 	69,60
45 		1,0099 		188,5 		188,4 	0,638 		4,182 	0,423 	637,3 	596,3 	68,78
50 		1,0121 		209,4 		209,3 	0,704 		4,181 	0,457 	643,6 	547,1 	67,95
60 		1,017089 		251,2 		251,1 	0,831 		4,183 	0,522 	654,4 	466,6 	66,24
70 		1,0227 		293,1 		293,0 	0,955 		4,187 	0,583 	663,1 	404,1 	64,49
80 		1,029027 		335,0 		334,9 	1,075 		4,194 	0,640 	670,0 	354,5 	62,68
90 		1,0359 		377,0 		376,9 	1,193 		4,204 	0,696 	675,3 	314,6 	60,82
99,63 	1,0431 		417,5 		417,4 	1,303 		4,217 	0,748 	679,0 	283,0 	58,99
100	1,043453		419,1

Stoffdaten von Wasser Quelle Wickipedia

*)
END_FUNCTION

(* POU WATER_ENTHALPY, ST *)
FUNCTION WATER_ENTHALPY : REAL
VAR_INPUT
	T : REAL;
END_VAR
VAR
	Pts : INT := 11;
	data : ARRAY[1..20, 0..1] OF REAL := 0,0.06, 10,42.1, 20,83.9, 30,125.8, 40,167.58, 50,209.4, 60,251.2, 70,293.1, 80,335.0, 90, 377.0, 100,419.1 ;
END_VAR

(*
version 1.0	29 oct 2007
programmer 	hugo
tested by		tobias

water_enthalpy calculates the enthalpy of liquid water from 0..100 °C 

*)
WATER_ENTHALPY := LINEAR_INT(T, Data, Pts);


(* revision history

hm	29.10.2007	rev 1.0
	original version

*)

(*
    °C - die Celsius-Temperatur in Grad Celsius
    v – das spezifische Volumen in Kubikdezimeter je Kilogramm dm³/kg
    h – die spezifische Enthalpie in Kilojoule je Kilogramm 	kJ/kg
    u – die spezifische Innere Energie in Kilojoule je Kilogramm 	kJ/kg
    s – die spezifische Entropie in Kilojoule je Kilogramm mal Kelvin 	kJ/(kg·K)
    cp - die spezifische Wärmekapazität bei konstantem Druck in Kilojoule je Kilogramm mal Kelvin 	kJ/(kg·K)
    Y – Volumenausdehnungskoeffizient in 10-3 durch Kelvin  10-3/K
    L – Wärmeleitfähigkeit in Milliwatt je Meter mal Kelvin  mW / (m·K) 
    n – Viskosität in Mikropascal mal Sekunde uPa·s 	
    s ? – Oberflächenspannung in Millinewton je Meter  mN/m


°C 		v 				h 			u 		s 			cp 		Y 		L		n		s	
-20		1,006580	
0 		1,000160 		0,06 		-0,04 	-0,0001 	4,228 	-0,080 	561,0 	1792 	75,65
4		1,000028
5 		1,0000 		21,1 		21,0 	0,076 		4,200 	0,011 	570,6 	1518 	74,95
10 		1,0003 		42,1 		42,0 	0,151 		4,188 	0,087 	580,0 	1306 	74,22
15 		1,0009 		63,0 		62,9 	0,224 		4,184 	0,152 	589,4 	1137 	73,49
20 		1,001797 		83,9 		83,8 	0,296 		4,183 	0,209 	598,4 	1001 	72,74
25 		1,0029 		104,8 		104,7 	0,367 		4,183 	0,259 	607,2 	890,4 	71,98
30 		1,0044 		125,8 		125,7 	0,437 		4,183 	0,305 	615,5 	797,7 	71,20
35 		1,0060 		146,7 		146,6 	0,505 		4,183 	0,347 	623,3 	719,6 	70,41
40 		1,007842 		167,58 	167,5 	0,572 		4,182 	0,386 	630,6 	653,3 	69,60
45 		1,0099 		188,5 		188,4 	0,638 		4,182 	0,423 	637,3 	596,3 	68,78
50 		1,0121 		209,4 		209,3 	0,704 		4,181 	0,457 	643,6 	547,1 	67,95
60 		1,017089 		251,2 		251,1 	0,831 		4,183 	0,522 	654,4 	466,6 	66,24
70 		1,0227 		293,1 		293,0 	0,955 		4,187 	0,583 	663,1 	404,1 	64,49
80 		1,029027 		335,0 		334,9 	1,075 		4,194 	0,640 	670,0 	354,5 	62,68
90 		1,0359 		377,0 		376,9 	1,193 		4,204 	0,696 	675,3 	314,6 	60,82
99,63 	1,0431 		417,5 		417,4 	1,303 		4,217 	0,748 	679,0 	283,0 	58,99
100	1,043453		419,1

Stoffdaten von Wasser Quelle Wickipedia

Wasser hat unter Normaldruck seine größte Dichte von 1000 Kilogramm pro Kubikmeter bei 3,98 °C und zeigt damit eine Dichteanomalie. 
Diese besteht darin, dass sich Wasser unterhalb von 3,98 °C bei weiterer Temperaturverringerung, auch beim Wechsel zum festen 
Aggregatzustand, wieder ausdehnt, was man nur von wenigen Stoffen kennt. Die derzeit genauesten publizierten Werte für die maximale 
Dichte liegen bei (999,974950 ± 0,00084) kg/m³ und bei (3,983 ± 0,00067) °C für die Temperatur, bei der dieser Wert erreicht wird. 
Die Werte stellen einen Mittelwert der von verschiedenen physikalischen Instituten veröffentlichten Zahlen dar (Stand 2001).

Die Berechnung der Dichte von luftfreiem Wasser DLF in Abhängigkeit von der Temperatur T ([T] = °C) kann mit Hilfe der folgenden 
Virialgleichung erfolgen:
: \frac{D_{\rm LF}}{\rm g/l} = \frac{a_0 + a_1 T + a_2 T^2 + a_3 T^3 + a_4 T^4 + a_5 T^5}{1 + b T}.
mit den Koeffizienten: a0 = 999,83952; a1 = 16,952577 (°C)-1; a2 = -7,9905127·10-3 (°C)-2; a3 = -4,6241757·10-5 (°C)-3; 
a4 = 1,0584601·10-7 (°C)-4; a5 = -2,8103006·10-10 (°C)-5 und b = 0,0168872. 
Für die Berechnung der Dichte von luftgesättigtem Wasser korrigiert man den Wert nach 
DLG/(g/l) = DLF/(g/l) - 0,004612 + 0,000106 (°C)-1·T. (Quelle: PTB-Mitteilungen 100/3-90)

*)
END_FUNCTION

(* POU LINEAR_INT, ST *)
FUNCTION LINEAR_INT : REAL
VAR_INPUT
	X : REAL;
	XY : ARRAY[1..20,0..1] OF REAL;
	Pts : INT;
END_VAR
VAR
	i : INT;
END_VAR

(*
	version 1.1	27 dec 2007
	programmer 	oscat
	tested BY		oscat

LINEAR_INT calculates an output based on a linear interpolation of up to 20 coordinates given in an array
the input coordinates have to start at the lowest array position and must be sorted ba ascending X values.

*)
(*make sure n is bound within the array size *)
pts := MIN(pts,20);

(* calculate the linear segement interpolation *)
i := 2;
(* search for segment and calculate output
	below and above the defined segments we interpolate the last segment *)
WHILE (i < pts) AND (XY[i,0] < X) DO
	i := i + 1;
END_WHILE;

(* calculate the output value on the corresponding segment coordinates *)
LINEAR_INT := ((XY[i,1] - XY[i-1,1]) * X - XY[i,1] * XY[i-1,0] + XY[i-1,1] * XY[i,0]) / (XY[i,0] - XY[i-1,0]);

(* revision history
hm	7. oct 2007		rev 1.0
	original version

hm	27 dec 2007		rev 1.1
	changed code for better performance
*)
END_FUNCTION

(* POU HEAT_TEMP, ST *)
FUNCTION_BLOCK HEAT_TEMP
VAR_INPUT
	T_EXT : REAL;
	T_INT : REAL;
	OFFSET : REAL;
	T_REQ : REAL;
END_VAR
VAR_INPUT CONSTANT
	TY_MAX : REAL := 70;
	TY_MIN : REAL := 25;
	TY_CONFIG : REAL := 70;
	T_INT_CONFIG : REAL := 20;
	T_EXT_CONFIG : REAL := -15;
	T_DIFF : REAL := 10;
	C : REAL := 1.33;
	H : REAL := 3;
END_VAR
VAR_OUTPUT
	TY : REAL;
	HEAT : BOOL;
END_VAR
VAR
	tr : REAL;
	tx: REAL;
END_VAR

(*
version 1.1	26. sep. 2008
programmer 	hugo
tested by	oscat

Heat_Temp calculates a heat characteristic based on the formula: tv=ti+(tvmax-ti)*((ti-tau)/(ti-taumin))^(1/n)
while
tv necessary heating temperature.
ti internal room temperature (20°C)
tau current external temperature
taumin external temperature to determine characteristics
C exponent for heating system (normally 1,33 or 1,1 for floor heating)

The two additional inputs TY_min and TY_max set limits for the output TY, while an offset inputs allows to rise or lower the room temperature.

*)
tr := T_INT + OFFSET;
tx := (tr - T_EXT) / (T_INT_CONFIG - T_EXT_CONFIG);

IF T_EXT + H > tr THEN
	TY := 0;
ELSE
	TY := LIMIT(TY_MIN, tr + T_DIFF / 2 * tx + (TY_CONFIG - T_DIFF/2 - tr) * EXPT(tx, 1 / C), TY_MAX);
END_IF;

TY := MAX(TY, T_REQ);
HEAT := TY > 0;


(*

tv=ti+(tvmax-ti)*((ti-tau)/(ti-taumin))^(1/n)

tv aktuelle Vorlauftemp.
ti Raumtemperatur innen (20°C)
tau aktuelle Außentemperatur
taumin minimale Außentemperatur -12°C oder -15°C
n Heizkörperexponent (meistens 1,33)
Fußbodenheizung = 1,1
Wandheizung 1,3

Normen z. B. DIN 4703, DIN 4725 oder die Literatur, z. B Recknagel Abschnitt 1.3.5.

*)


(* revision history
hm	27. jan. 2008	rev 1.0
	original version

hm	26. sep. 2008	rev 1.1
	moved T_INT from config to Input
	added config variable H
	corrected error in formula
*)
END_FUNCTION_BLOCK

(* POU HOUR_OF_DT, ST *)
FUNCTION HOUR_OF_DT : INT
VAR_INPUT
	XDT : DT;
END_VAR
VAR
END_VAR


(*
	version 1.0	6. jun. 2008
	programmer 	oscat
	tested BY	oscat

HOUR_OF_DT returns the current hour (hour of the day) of a DT variable

*)
HOUR_OF_DT := DWORD_TO_INT((DT_TO_DWORD(XDT) MOD 86400)/3600);


(* revision history
hm		6.9.2008	rev 1.0
	original version


*)
END_FUNCTION

(* POU HOUR_TO_TIME, ST *)
FUNCTION HOUR_TO_TIME : TIME
VAR_INPUT
	input : REAL;
END_VAR
VAR
END_VAR

(*
version 1.1	14 mar 2008
programmer 	hugo
tested by		tobias

converts an amount of hours in real to time

*)
hour_to_time := DWORD_TO_TIME(REAL_TO_DWORD(input * 3600000));


(* revision history
hm		4. aug 2006	rev 1.0
	original version

hm		14. mar 2008	rev 1.1
	rounded the input after the last digit

*)
END_FUNCTION

